METHOD PRIVATE CheckCanHomeTransferArm
VAR_IN_OUT
    stSDS : ST_SDS;
    stSDSP : ST_SDSPersistent;
END_VAR

stSDS.bSuccess := FALSE;

stSDS.sStatusMsg := 'Checking if transfer arm can be homed.';

InitHomeTransferArm(
    stSDS := stSDS
);

stSDS.bSuccess := TRUE;
END_METHOD


METHOD PRIVATE CheckCanLoadArmFromGarage
VAR_IN_OUT
    stSDS : ST_SDS;
    stSDSP : ST_SDSPersistent;
END_VAR

stSDS.bSuccess := FALSE;

stSDS.sStatusMsg := 'Checking if there is an open slot in the transfer arm and at least one full slot in the garage.';

CheckCanDo2Criteria(
    bCanDo := stSDS.bSuccess,
    bCantDo := stSDS.bError,
    sErrorMsg := stSDS.sErrorMsg,
    b1 := stSDS.bGarageUnloadable,
    b2 := stSDS.bTransferArmLoadable,
    sErrorMsgTF := 'The transfer arm is currently full and cannot be used to remove a sample from the garage.',
    sErrorMsgFT := 'The garage is currently empty and therefore no samples can be removed.',
    sErrorMsgFF := 'The garage is currently empty and the transfer arm is full. Therefore, no samples can be removed.'
);
END_METHOD


METHOD PRIVATE CheckCanLoadDiffractometerFromArm
VAR_IN_OUT
    stSDS : ST_SDS;
    stSDSP : ST_SDSPersistent;
END_VAR

stSDS.bSuccess := FALSE;

stSDS.sStatusMsg := 'Checking if the diffractometer slot is open and if the transfer arm is carrying a sample.';

CheckCanDo2Criteria(
    bCanDo := stSDS.bSuccess,
    bCantDo := stSDS.bError,
    sErrorMsg := stSDS.sErrorMsg,
    b1 := stSDS.bDiffractometerLoadable,
    b2 := stSDS.bTransferArmUnloadable,
    sErrorMsgTF := 'The transfer arm is currently empty and cannot be used to place a sample in the diffractometer.',
    sErrorMsgFT := 'The diffractometer already has a sample in it.',
    sErrorMsgFF := 'The diffractoemter already has a sample and the transfer arm is empty.'
);
END_METHOD


METHOD PRIVATE CheckCanLoadUnloadGarageFromPort
VAR_IN_OUT
    stSDS : ST_SDS;
    stSDSP : ST_SDSPersistent;
END_VAR

stSDS.bSuccess := FALSE;

stSDS.sStatusMsg := 'Checking if the garage can be loaded or unloaded from the port.';

stSDS.bSuccess := TRUE;
END_METHOD


METHOD PRIVATE CheckCanManualControl
VAR_IN_OUT
    stSDS : ST_SDS;
    stSDSP : ST_SDSPersistent;
END_VAR

stSDS.bSuccess := FALSE;

stSDS.sStatusMsg := 'Checking if we can switch to manual control.';

stSDS.bSuccess := TRUE;
END_METHOD


METHOD PRIVATE CheckCanUnloadArmToGarage
VAR_IN_OUT
    stSDS : ST_SDS;
    stSDSP : ST_SDSPersistent;
END_VAR

stSDS.bSuccess := FALSE;

stSDS.sStatusMsg := 'Checking if there is an open slot in the garage and if the transfer arm is carrying a sample.';

CheckCanDo2Criteria(
    bCanDo := stSDS.bSuccess,
    bCantDo := stSDS.bError,
    sErrorMsg := stSDS.sErrorMsg,
    b1 := stSDS.bGarageLoadable,
    b2 := stSDS.bTransferArmUnloadable,
    sErrorMsgTF := 'The transfer arm is currently empty and cannot be used to load sample into the garage.',
    sErrorMsgFT := 'The garage is currently full and therefore no samples can be loaded into it.',
    sErrorMsgFF := 'The garage is currently full and the transfer arm is empty.'
);
END_METHOD


METHOD PRIVATE CheckCanUnloadDiffractometerToArm
VAR_IN_OUT
    stSDS : ST_SDS;
    stSDSP : ST_SDSPersistent;
END_VAR

stSDS.bSuccess := FALSE;

stSDS.sStatusMsg := 'Checking if the diffractometer slot is full and if the transfer arm is empty.';

CheckCanDo2Criteria(
    bCanDo := stSDS.bSuccess,
    bCantDo := stSDS.bError,
    sErrorMsg := stSDS.sErrorMsg,
    b1 := stSDS.bDiffractometerUnloadable,
    b2 := stSDS.bTransferArmLoadable,
    sErrorMsgTF := 'The transfer arm is currently full and cannot be used to unload a sample from the diffractometer.',
    sErrorMsgFT := 'The diffractometer does not have a sample in it.',
    sErrorMsgFF := 'The diffractometeris empty and the transfer arm is full.'
);
END_METHOD


METHOD PRIVATE ConfirmDiffractometerExtraction
VAR_IN_OUT
    stSDS : ST_SDS;
END_VAR

stSDS.bSuccess := FALSE;

stSDS.sStatusMsg := 'Moving transfer arm back a few mm. Please confirm the sample is held by the diffractometer and then click "proceed". If the sample is still in the transfer arm, click "retry" to go back to fine adjustment.';

SetPositionStateWaitForArrivalQuitIfError(
    eStateGet := stSDS.eTransferArmHStateGet,
    stMotionStage := stSDS.stTransferArmHStage,
    eStateSet := stSDS.eTransferArmHStateSet,
    eEnumSet := E_SDSTransferArmHStates.CONFIRM_DIFF_EXTRACTION,
    bError := stSDS.bError,
    sErrorMsg := stSDS.sErrorMsg,
    bArrived => stSDS.bSuccess
);
END_METHOD


METHOD PRIVATE ConfirmDiffractometerInsertion
VAR_IN_OUT
    stSDS : ST_SDS;
END_VAR

stSDS.bSuccess := FALSE;

stSDS.sStatusMsg := 'Moving transfer arm back a few mm. Please confirm the sample is held by the diffractometer and then click "proceed". If the sample is still in the transfer arm, click "retry" to go back to fine adjustment.';

SetPositionStateWaitForArrivalQuitIfError(
    eStateGet := stSDS.eTransferArmHStateGet,
    stMotionStage := stSDS.stTransferArmHStage,
    eStateSet := stSDS.eTransferArmHStateSet,
    eEnumSet := E_SDSTransferArmHStates.CONFIRM_DIFF_INSERTION,
    bError := stSDS.bError,
    sErrorMsg := stSDS.sErrorMsg,
    bArrived => stSDS.bSuccess
);
END_METHOD


METHOD PRIVATE ConfirmExtraction
VAR_IN_OUT
    stSDS : ST_SDS;
END_VAR

stSDS.bSuccess := FALSE;

stSDS.sStatusMsg := 'Moving transfer arm back a few mm. Please confirm the sample is held by the arm and then click "proceed". If the sample is still in the holder, click "retry" to go back to fine adjustment.';

SetPositionStateWaitForArrivalQuitIfError(
    eStateGet := stSDS.eTransferArmHStateGet,
    stMotionStage := stSDS.stTransferArmHStage,
    eStateSet := stSDS.eTransferArmHStateSet,
    eEnumSet := E_SDSTransferArmHStates.CONFIRM_GARAGE_EXTRACTION,
    bError := stSDS.bError,
    sErrorMsg := stSDS.sErrorMsg,
    bArrived => stSDS.bSuccess
);
END_METHOD


METHOD PRIVATE ConfirmGarageFreeToRotate
VAR_IN_OUT
    stSDS : ST_SDS;
    stSDSP : ST_SDSPersistent;
END_VAR
VAR_INST
    tonHoldDelay : TON;
END_VAR

// Missing handling for erroring encoder.

tonHoldDelay(
    IN := stSDS.stGarageYStage.Axis.NcToPlc.ActPos >= stSDSP.fGarageHeightSafeFromCollision,
    PT := T#1s
);

stSDS.bGarageAboveCollisionHeight := tonHoldDelay.Q;
END_METHOD


METHOD PRIVATE ConfirmInsertion
VAR_IN_OUT
    stSDS : ST_SDS;
END_VAR

stSDS.bSuccess := FALSE;

stSDS.sStatusMsg := 'Moving transfer arm back a few mm. Please confirm the sample is held by the garage and then click "proceed". If the sample is still in the transfer arm, click "retry" to go back to fine adjustment.';

SetPositionStateWaitForArrivalQuitIfError(
    eStateGet := stSDS.eTransferArmHStateGet,
    stMotionStage := stSDS.stTransferArmHStage,
    eStateSet := stSDS.eTransferArmHStateSet,
    eEnumSet := E_SDSTransferArmHStates.CONFIRM_GARAGE_INSERTION,
    bError := stSDS.bError,
    sErrorMsg := stSDS.sErrorMsg,
    bArrived => stSDS.bSuccess
);
END_METHOD


METHOD PRIVATE ConfirmVacuumValveOpen
VAR_IN_OUT
    stSDS : ST_SDS;
END_VAR

stSDS.sStatusMsg := 'Verifying that the vacuum valve between SDS and Diff is open.';

stSDS.bSuccess := GVL_Interface.QRIX_VAC_VGC_03_OPEN_LIMIT_SWITCH AND
    NOT GVL_Interface.QRIX_VAC_VGC_03_CLOSED_LIMIT_SWITCH;
END_METHOD


METHOD PRIVATE ExtendPrerotateTransferArmForLoading
VAR_IN_OUT
    stSDS : ST_SDS;
END_VAR
VAR
    bHArrived : BOOL;
    bRArrived : BOOL;
END_VAR

stSDS.bSuccess := FALSE;

stSDS.sStatusMsg := 'Moving transfer arm to nominal sample loading position and pre-rotating to allow full rotation for screwing in sample.';

SetPositionStateWaitForArrivalQuitIfError(
    eStateGet := stSDS.eTransferArmHStateGet,
    stMotionStage := stSDS.stTransferArmHStage,
    eStateSet := stSDS.eTransferArmHStateSet,
    eEnumSet := E_SDSTransferArmHStates.GARAGE_SAMPLE_INSERTION,
    bError := stSDS.bError,
    sErrorMsg := stSDS.sErrorMsg,
    bArrived => bHArrived
);

SetPositionStateWaitForArrivalQuitIfError(
    eStateGet := stSDS.eTransferArmRStateGet,
    stMotionStage := stSDS.stTransferArmRStage,
    eStateSet := stSDS.eTransferArmRStateSet,
    eEnumSet := E_SDSTransferArmRStates.PREROTATE_SAMPLE_INSERTION,
    bError := stSDS.bError,
    sErrorMsg := stSDS.sErrorMsg,
    bArrived => bRArrived
);

IF bHArrived AND bRArrived THEN
    stSDS.bSuccess := TRUE;
END_IF
END_METHOD


METHOD PRIVATE ExtendTransferArmForDiffractometerExtraction
VAR_IN_OUT
    stSDS : ST_SDS;
END_VAR

stSDS.bSuccess := FALSE;

stSDS.sStatusMsg := 'Moving transfer arm to nominal sample unloading position for diffractometer.';

SetPositionStateWaitForArrivalQuitIfError(
    eStateGet := stSDS.eTransferArmHStateGet,
    stMotionStage := stSDS.stTransferArmHStage,
    eStateSet := stSDS.eTransferArmHStateSet,
    eEnumSet := E_SDSTransferArmHStates.DIFF_SAMPLE_EXTRACTION,
    bError := stSDS.bError,
    sErrorMsg := stSDS.sErrorMsg,
    bArrived => stSDS.bSuccess
);
END_METHOD


METHOD PRIVATE ExtendTransferArmForDiffractometerInsertion
VAR_IN_OUT
    stSDS : ST_SDS;
END_VAR

stSDS.bSuccess := FALSE;

stSDS.sStatusMsg := 'Moving transfer arm to nominal sample loading position for diffractometer.';

SetPositionStateWaitForArrivalQuitIfError(
    eStateGet := stSDS.eTransferArmHStateGet,
    stMotionStage := stSDS.stTransferArmHStage,
    eStateSet := stSDS.eTransferArmHStateSet,
    eEnumSet := E_SDSTransferArmHStates.DIFF_SAMPLE_INSERTION,
    bError := stSDS.bError,
    sErrorMsg := stSDS.sErrorMsg,
    bArrived => stSDS.bSuccess
);
END_METHOD


METHOD PRIVATE ExtendTransferArmForExtraction
VAR_IN_OUT
    stSDS : ST_SDS;
END_VAR

stSDS.bSuccess := FALSE;

stSDS.sStatusMsg := 'Moving transfer arm to nominal sample extraction position for garage.';

SetPositionStateWaitForArrivalQuitIfError(
    eStateGet := stSDS.eTransferArmHStateGet,
    stMotionStage := stSDS.stTransferArmHStage,
    eStateSet := stSDS.eTransferArmHStateSet,
    eEnumSet := E_SDSTransferArmHStates.GARAGE_SAMPLE_REMOVAL,
    bError := stSDS.bError,
    sErrorMsg := stSDS.sErrorMsg,
    bArrived => stSDS.bSuccess
);
END_METHOD


METHOD PRIVATE ExtendTransferArmForInsertion
VAR_IN_OUT
    stSDS : ST_SDS;
END_VAR
VAR
    bHArrived : BOOL;
    bRArrived : BOOL;
END_VAR

stSDS.bSuccess := FALSE;

stSDS.sStatusMsg := 'Moving transfer arm to nominal sample loading position for garage.';

SetPositionStateWaitForArrivalQuitIfError(
    eStateGet := stSDS.eTransferArmHStateGet,
    stMotionStage := stSDS.stTransferArmHStage,
    eStateSet := stSDS.eTransferArmHStateSet,
    eEnumSet := E_SDSTransferArmHStates.GARAGE_SAMPLE_INSERTION,
    bError := stSDS.bError,
    sErrorMsg := stSDS.sErrorMsg,
    bArrived => stSDS.bSuccess
);
END_METHOD


METHOD PRIVATE FineAdjustment
VAR_IN_OUT
    stSDS : ST_SDS;
END_VAR

stSDS.sStatusMsg := 'Use the individual motor control to do fine adjustment. Click "proceed" to move to the next step.';
END_METHOD


METHOD PRIVATE GarageFaceTransferArm
VAR_IN_OUT
    stSDS : ST_SDS;
END_VAR
VAR
    bYArrived : BOOL;
    bRArrived : BOOL;
END_VAR

stSDS.bSuccess := FALSE;

stSDS.sStatusMsg := 'Facing garage towards the transfer arm.';

stSDS.eFaceState := E_SDSFaceState.FACE_TRANSFER_ARM;

SetPositionStateWaitForArrivalQuitIfError(
    eStateGet := stSDS.eGarageRStateGet,
    stMotionStage := stSDS.stGarageRStage,
    eStateSet := stSDS.eGarageRStateSet,
    eEnumSet := stSDS.eSelectedGarageSlot,
    bError := stSDS.bError,
    sErrorMsg := stSDS.sErrorMsg,
    bArrived => stSDS.bSuccess
);
END_METHOD


METHOD PRIVATE HoldThenClear
VAR_IN_OUT
    b1 : BOOL;
END_VAR
VAR_INPUT
    tHoldDuration : TIME := T#1s;
END_VAR
VAR_INST
    tonHoldTimer : TON;
END_VAR

tonHoldTimer(IN := b1, PT := tHoldDuration);

IF tonHoldTimer.Q THEN
    b1 := FALSE;
END_IF
END_METHOD


METHOD PRIVATE HomeGarage
VAR_IN_OUT
    stSDS : ST_SDS;
END_VAR

stSDS.bSuccess := FALSE;

stSDS.sStatusMsg := 'Homing the garage.';

IF stSDS.stGarageRStage.bError THEN
    stSDS.bError := TRUE;
    stSDS.sErrorMsg := 'Garage rotational stage has an active error. Aborting sequence.';
END_IF

HomeStateMachine(
    eHomingState := stSDS.eGarageRHomingState,
    stMotionStage := stSDS.stGarageRStage,
    bError => stSDS.bError,
    sErrorMsg => stSDS.sErrorMsg
);

IF stSDS.eGarageRHomingState = E_SDSHomingState.HOMED THEN
    stSDS.bSuccess := TRUE;
END_IF
END_METHOD


METHOD PRIVATE HomeStateMachine
VAR_IN_OUT
    eHomingState : E_SDSHomingState;
    stMotionStage : ST_MotionStage;
END_VAR
VAR_OUTPUT
    bError : BOOL;
    sErrorMsg : T_MaxString;
END_VAR

IF stMotionStage.bHome AND F_Limit(
    fVal := stMotionStage.Axis.NcToPlc.ActPos,
    fLLim := -0.01,
    fHLim := 0.01,
    bInclusive := TRUE) THEN
    eHomingState := E_SDSHomingState.HOMED;
END_IF

CASE eHomingState OF
    E_SDSHomingState.INIT:
        eHomingState := E_SDSHomingState.WAIT_NOT_BUSY;
    E_SDSHomingState.WAIT_NOT_BUSY:
        IF NOT stMotionStage.bBusy THEN
            eHomingState := E_SDSHomingState.TRIGGER_HOMING;
        END_IF
    E_SDSHomingState.TRIGGER_HOMING:
        stMotionStage.bHomeCmd := TRUE;
        IF stMotionStage.nCommand = E_EpicsMotorCmd.HOME AND stMotionStage.bBusy THEN
            eHomingState := E_SDSHomingState.WAIT_FOR_HOMED;
        END_IF
    E_SDSHomingState.WAIT_FOR_HOMED:
        IF stMotionStage.bDone THEN
            eHomingState := E_SDSHomingState.HOMED;
        END_IF
ELSE
    bError := TRUE;
    sErrorMsg := 'Homing sequence triggered an unknown state. Aborting sequence.';
END_CASE
END_METHOD


METHOD PRIVATE HomeTransferArm
VAR_IN_OUT
    stSDS : ST_SDS;
END_VAR

stSDS.bSuccess := FALSE;

stSDS.sStatusMsg := 'Homing the transfer arm.';

IF stSDS.stTransferArmHStage.bError THEN
    stSDS.bError := TRUE;
    stSDS.sErrorMsg := 'Transfer arm horizontal stage has an active error. Aborting sequence.';
END_IF

IF stSDS.stTransferArmRStage.bError THEN
    stSDS.bError := TRUE;
    stSDS.sErrorMsg := 'Transfer arm rotational stage has an active error. Aborting sequence.';
END_IF

HomeStateMachine(
    eHomingState := stSDS.eTransferArmHHomingState,
    stMotionStage := stSDS.stTransferArmHStage,
    bError => stSDS.bError,
    sErrorMsg => stSDS.sErrorMsg
);

HomeStateMachine(
    eHomingState := stSDS.eTransferArmRHomingState,
    stMotionStage := stSDS.stTransferArmRStage,
    bError => stSDS.bError,
    sErrorMsg => stSDS.sErrorMsg
);

IF stSDS.eTransferArmHHomingState = E_SDSHomingState.HOMED AND
   stSDS.eTransferArmRHomingState = E_SDSHomingState.HOMED THEN
    stSDS.bSuccess := TRUE;
END_IF
END_METHOD


METHOD PRIVATE InitHomeGarage
VAR_IN_OUT
    stSDS : ST_SDS;
END_VAR

stSDS.eGarageRHomingState := E_SDSHomingState.INIT;
END_METHOD


METHOD PRIVATE InitHomeTransferArm
VAR_IN_OUT
    stSDS : ST_SDS;
END_VAR

stSDS.eTransferArmHHomingState := E_SDSHomingState.INIT;
stSDS.eTransferArmRHomingState := E_SDSHomingState.INIT;
END_METHOD


METHOD PRIVATE InitRotateGarageForClearance
VAR_IN_OUT
    stSDS : ST_SDS;
    stSDSP : ST_SDSPersistent;
END_VAR

stSDS.fGarageRotationClearancePos := stSDS.stGarageRStage.Axis.NcToPlc.ActPos + stSDSP.fGarageRotationClearanceOffset;
END_METHOD


METHOD PRIVATE InitSelectGarageSlotForLoading
VAR_IN_OUT
    stSDS : ST_SDS;
    stSDSP : ST_SDSPersistent;
END_VAR

FOR nIndex := E_SDSGarageYStates.T1 TO E_SDSGarageYStates.B4 BY 1 DO
    CASE stSDSP.astGarageSlot[nIndex].eState OF
        E_SampleSlotStates.EMPTY:
            stSDS.eSelectedGarageSlot := nIndex;
    END_CASE
END_FOR

IF nIndex > E_SDSGarageYStates.B4 THEN
    stSDS.bError := TRUE;
    stSDS.sErrorMsg := 'There are no empty slots in the garage to load a sample to.';
END_IF
END_METHOD


METHOD PRIVATE InitSelectGarageSlotForRemoval
VAR_IN_OUT
    stSDS : ST_SDS;
    stSDSP : ST_SDSPersistent;
END_VAR

FOR nIndex := E_SDSGarageYStates.T1 TO E_SDSGarageYStates.B4 BY 1 DO
    CASE stSDSP.astGarageSlot[nIndex].eState OF
        E_SampleSlotStates.FULL:
            stSDS.eSelectedGarageSlot := nIndex;
    END_CASE
END_FOR

IF nIndex > E_SDSGarageYStates.B4 THEN
    stSDS.bError := TRUE;
    stSDS.sErrorMsg := 'There are no full slots in the garage to extract a sample from.';
END_IF
END_METHOD


METHOD PRIVATE LoadArmFromGarage
VAR_IN_OUT
    stSDS : ST_SDS;
    stSDSP : ST_SDSPersistent;
END_VAR

CASE stSDS.eSeqState OF
    E_SDSSeqState.Inactive:
        stSDS.eSeqState := E_SDSSeqState.Home_Transfer_Arm;
    E_SDSSeqState.Home_Transfer_Arm:
        HomeTransferArm(
            stSDS := stSDS
        );
        IF stSDS.bSuccess THEN
            stSDS.eSeqState := E_SDSSeqState.Check_Garage_Height;
        END_IF
    E_SDSSeqState.Check_Garage_Height:
        IF stSDS.bGarageAboveCollisionHeight THEN
            stSDS.eSeqState := E_SDSSeqState.Home_Garage;
        ELSE
            stSDS.eSeqState := E_SDSSeqState.Manually_Rotate_Garage_for_Clearance_to_Raise;
        END_IF
    E_SDSSeqState.Manually_Rotate_Garage_for_Clearance_to_Raise:
        RotateGarageForClearanceManual(
            stSDS := stSDS
        );
        IF stSDS.stUISelect.bProceed THEN
            stSDS.eSeqState := E_SDSSeqState.Retract_Garage_1;
        END_IF
    E_SDSSeqState.Retract_Garage_1:
        RetractGarage(
            stSDS := stSDS
        );
        IF stSDS.bSuccess THEN
            stSDS.eSeqState := E_SDSSeqState.Home_Garage;
        END_IF
    E_SDSSeqState.Home_Garage:
        HomeGarage(
            stSDS := stSDS
        );
        IF stSDS.bSuccess THEN
            stSDS.eSeqState := E_SDSSeqState.Select_Garage_Slot_for_Removal;
        END_IF
    E_SDSSeqState.Select_Garage_Slot_for_Removal:
        SelectGarageSlotForRemoval(
            stSDS := stSDS,
            stSDSP := stSDSP
        );
        IF stSDS.bSuccess THEN
            stSDS.eSeqState := E_SDSSeqState.Garage_Face_Transfer_Arm;
        END_IF
    E_SDSSeqState.Garage_Face_Transfer_Arm:
        GarageFaceTransferArm(
            stSDS := stSDS
        );
        IF stSDS.bSuccess THEN
            stSDS.eSeqState := E_SDSSeqState.Rotate_Garage_for_Clearance_to_Lower;
        END_IF
    E_SDSSeqState.Rotate_Garage_for_Clearance_to_Lower:
        RotateGarageForClearance(
            stSDS := stSDS
        );
        IF stSDS.bSuccess THEN
            stSDS.eSeqState := E_SDSSeqState.Move_Garage_to_Slot_Height;
        END_IF
    E_SDSSeqState.Move_Garage_to_Slot_Height:
        MoveGarageToSlotHeight(
            stSDS := stSDS
        );
        IF stSDS.bSuccess THEN
            stSDS.eSeqState := E_SDSSeqState.Prerotate_Transfer_Arm_for_Extraction;
        END_IF
    E_SDSSeqState.Prerotate_Transfer_Arm_for_Extraction:
        PrerotateTransferArmForExtraction(
            stSDS := stSDS
        );
        IF stSDS.bSuccess THEN
            stSDS.eSeqState := E_SDSSeqState.Extend_Transfer_Arm_for_Extraction;
        END_IF
    E_SDSSeqState.Extend_Transfer_Arm_for_Extraction:
        ExtendTransferArmForExtraction(
            stSDS := stSDS
        );
        IF stSDS.bSuccess THEN
            stSDS.eSeqState := E_SDSSeqState.Screw_in_Half_Turn;
        END_IF
    E_SDSSeqState.Screw_in_Half_Turn:
        ScrewInHalfTurn(
            stSDS := stSDS
        );
        IF stSDS.bSuccess THEN
            stSDS.eSeqState := E_SDSSeqState.Fine_Adjustment;
        END_IF
    E_SDSSeqState.Fine_Adjustment:
        FineAdjustment(
            stSDS := stSDS
        );
        IF stSDS.stUISelect.bProceed THEN
            stSDS.eSeqState := E_SDSSeqState.Unscrew_Sample_from_Garage;
        END_IF
    E_SDSSeqState.Unscrew_Sample_from_Garage:
        UnscrewSampleFromGarage(
            stSDS := stSDS
        );
        IF stSDS.bSuccess THEN
            stSDS.eSeqState := E_SDSSeqState.Confirm_Extraction;
        END_IF
    E_SDSSeqState.Confirm_Extraction:
        ConfirmExtraction(
            stSDS := stSDS
        );
        IF stSDS.bSuccess AND stSDS.stUISelect.bProceed THEN
            stSDS.eSeqState := E_SDSSeqState.Update_Sample_Database;
        ELSIF stSDS.stUISelect.bRetry THEN
            stSDS.eSeqState := E_SDSSeqState.Fine_Adjustment;
        END_IF
    E_SDSSeqState.Update_Sample_Database:
        UpdateSampleLocationDatabaseGarageToArm(
            stSDS := stSDS,
            stSDSP := stSDSP
        );
        IF stSDS.bSuccess OR stSDS.stUISelect.bProceed THEN
            stSDS.eSeqState := E_SDSSeqState.Retract_Transfer_Arm;
        END_IF
    E_SDSSeqState.Retract_Transfer_Arm:
        HomeTransferArm(
            stSDS := stSDS
        );
        IF stSDS.bSuccess THEN
            stSDS.eSeqState := E_SDSSeqState.Rotate_Garage_for_Clearance_to_Raise;
        END_IF
    E_SDSSeqState.Rotate_Garage_for_Clearance_to_Raise:
        RotateGarageForClearance(
            stSDS := stSDS
        );
        IF stSDS.bSuccess THEN
            stSDS.eSeqState := E_SDSSeqState.Retract_Garage_2;
        END_IF
    E_SDSSeqState.Retract_Garage_2:
        RetractGarage(
            stSDS := stSDS
        );
        IF stSDS.bSuccess THEN
            stSDS.eSeqState := E_SDSSeqState.Return_Garage_to_Home;
        END_IF
    E_SDSSeqState.Return_Garage_to_Home:
        HomeGarage(
            stSDS := stSDS
        );
        IF stSDS.bSuccess THEN
            stSDS.eState := E_SDSState.Standby;
        END_IF
END_CASE
END_METHOD


METHOD PRIVATE LoadDiffractometerFromArm
VAR_IN_OUT
    stSDS : ST_SDS;
    stSDSP : ST_SDSPersistent;
END_VAR

CASE stSDS.eSeqState OF
    E_SDSSeqState.Inactive:
        stSDS.eSeqState := E_SDSSeqState.Home_Transfer_Arm;
    E_SDSSeqState.Home_Transfer_Arm:
        HomeTransferArm(
            stSDS := stSDS
        );
        IF stSDS.bSuccess THEN
            stSDS.eSeqState := E_SDSSeqState.Check_Garage_Height;
        END_IF
    E_SDSSeqState.Check_Garage_Height:
        IF stSDS.bGarageAboveCollisionHeight THEN
            stSDS.eSeqState := E_SDSSeqState.Home_Garage;
        ELSE
            stSDS.eSeqState := E_SDSSeqState.Manually_Rotate_Garage_for_Clearance_to_Raise;
        END_IF
    E_SDSSeqState.Manually_Rotate_Garage_for_Clearance_to_Raise:
        RotateGarageForClearanceManual(
            stSDS := stSDS
        );
        IF stSDS.stUISelect.bProceed THEN
            stSDS.eSeqState := E_SDSSeqState.Retract_Garage_1;
        END_IF
    E_SDSSeqState.Retract_Garage_1:
        RetractGarage(
            stSDS := stSDS
        );
        IF stSDS.bSuccess THEN
            stSDS.eSeqState := E_SDSSeqState.Home_Garage;
        END_IF
    E_SDSSeqState.Home_Garage:
        HomeGarage(
            stSDS := stSDS
        );
        IF stSDS.bSuccess THEN
            stSDS.eSeqState := E_SDSSeqState.Move_Diffractometer_to_Load_Unload_Position;
        END_IF
    E_SDSSeqState.Move_Diffractometer_to_Load_Unload_Position:
        MoveDiffractometerToLoadUnloadPosition(
            stSDS := stSDS
        );
        IF stSDS.bSuccess THEN
            stSDS.eSeqState := E_SDSSeqState.Confirm_Vacuum_Valve_Open;
        END_IF
    E_SDSSeqState.Confirm_Vacuum_Valve_Open:
        ConfirmVacuumValveOpen(
            stSDS := stSDS
        );
        IF stSDS.bSuccess THEN
            stSDS.eSeqState := E_SDSSeqState.Prerotate_Transfer_Arm_for_Insertion;
        END_IF
    E_SDSSeqState.Prerotate_Transfer_Arm_for_Insertion:
        PrerotateTransferArmForInsertion(
            stSDS := stSDS
        );
        IF stSDS.bSuccess THEN
            stSDS.eSeqState := E_SDSSeqState.Extend_Transfer_Arm_for_Diffractometer_Insertion;
        END_IF
    E_SDSSeqState.Extend_Transfer_Arm_for_Diffractometer_Insertion:
        ExtendTransferArmForDiffractometerInsertion(
            stSDS := stSDS
        );
        IF stSDS.bSuccess THEN
            stSDS.eSeqState := E_SDSSeqState.Fine_Adjustment;
        END_IF
    E_SDSSeqState.Fine_Adjustment:
        FineAdjustment(
            stSDS := stSDS
        );
        IF stSDS.stUISelect.bProceed THEN
            stSDS.eSeqState := E_SDSSeqState.Screw_Sample_into_Diffractometer;
        END_IF
    E_SDSSeqState.Screw_Sample_into_Diffractometer:
        ScrewSampleIntoDiffractometer(
            stSDS := stSDS
        );
        IF stSDS.bSuccess THEN
            stSDS.eSeqState := E_SDSSeqState.Confirm_Diffractometer_Insertion;
        END_IF
    E_SDSSeqState.Confirm_Diffractometer_Insertion:
        ConfirmDiffractometerInsertion(
            stSDS := stSDS
        );
        IF stSDS.bSuccess AND stSDS.stUISelect.bProceed THEN
            stSDS.eSeqState := E_SDSSeqState.Update_Sample_Database;
        ELSIF stSDS.stUISelect.bRetry THEN
            stSDS.eSeqState := E_SDSSeqState.Fine_Adjustment;
        END_IF
    E_SDSSeqState.Update_Sample_Database:
        UpdateSampleLocationDatabaseDiffToArm(
            stSDS := stSDS,
            stSDSP := stSDSP
        );
        IF stSDS.bSuccess OR stSDS.stUISelect.bProceed THEN
            stSDS.eSeqState := E_SDSSeqState.Retract_Transfer_Arm;
        END_IF
    E_SDSSeqState.Retract_Transfer_Arm:
        HomeTransferArm(
            stSDS := stSDS
        );
        IF stSDS.bSuccess THEN
            stSDS.eSeqState := E_SDSSeqState.Rotate_Garage_for_Clearance_to_Raise;
        END_IF
END_CASE
END_METHOD


METHOD PRIVATE LoadUnloadGarageFromPort
VAR_IN_OUT
    stSDS : ST_SDS;
    stSDSP : ST_SDSPersistent;
END_VAR
END_METHOD


METHOD PRIVATE ManualControl
VAR_IN_OUT
    stSDS : ST_SDS;
    stSDSP : ST_SDSPersistent;
END_VAR
END_METHOD


METHOD PRIVATE MoveDiffractometerToLoadUnloadPosition
VAR_IN_OUT
    stSDS : ST_SDS;
END_VAR
VAR
    bXArrived : BOOL;
    bYArrived : BOOL;
    bZArrived : BOOL;
    b2ThetaYArrived : BOOL;
    bPhiArrived : BOOL;
    bChiArrived : BOOL;
    b2ThetaArrived : BOOL;
    bThetaArrived : BOOL;
END_VAR

stSDS.bSuccess := FALSE;

stSDS.sStatusMsg := 'Moving the diffractometer to load/unload position.';

SetPositionStateWaitForArrivalQuitIfError(
    eStateGet := stSDS.eDiffXStateGet,
    stMotionStage := stSDS.stDiffXStage,
    eStateSet := stSDS.eDiffXStateSet,
    eEnumSet := E_DiffState.TRANSFER_ARM_INTERFACE,
    bError := stSDS.bError,
    sErrorMsg := stSDS.sErrorMsg,
    bArrived => bXArrived
);

SetPositionStateWaitForArrivalQuitIfError(
    eStateGet := stSDS.eDiffYStateGet,
    stMotionStage := stSDS.stDiffYStage,
    eStateSet := stSDS.eDiffYStateSet,
    eEnumSet := E_DiffState.TRANSFER_ARM_INTERFACE,
    bError := stSDS.bError,
    sErrorMsg := stSDS.sErrorMsg,
    bArrived => bYArrived
);

SetPositionStateWaitForArrivalQuitIfError(
    eStateGet := stSDS.eDiffZStateGet,
    stMotionStage := stSDS.stDiffZStage,
    eStateSet := stSDS.eDiffZStateSet,
    eEnumSet := E_DiffState.TRANSFER_ARM_INTERFACE,
    bError := stSDS.bError,
    sErrorMsg := stSDS.sErrorMsg,
    bArrived => bZArrived
);

SetPositionStateWaitForArrivalQuitIfError(
    eStateGet := stSDS.eDiff2ThetaYStateGet,
    stMotionStage := stSDS.stDiff2ThetaYStage,
    eStateSet := stSDS.eDiff2ThetaYStateSet,
    eEnumSet := E_DiffState.TRANSFER_ARM_INTERFACE,
    bError := stSDS.bError,
    sErrorMsg := stSDS.sErrorMsg,
    bArrived => b2ThetaYArrived
);

SetPositionStateWaitForArrivalQuitIfError(
    eStateGet := stSDS.eDiffPhiStateGet,
    stMotionStage := stSDS.stDiffPhiStage,
    eStateSet := stSDS.eDiffPhiStateSet,
    eEnumSet := E_DiffState.TRANSFER_ARM_INTERFACE,
    bError := stSDS.bError,
    sErrorMsg := stSDS.sErrorMsg,
    bArrived => bPhiArrived
);

SetPositionStateWaitForArrivalQuitIfError(
    eStateGet := stSDS.eDiffChiStateGet,
    stMotionStage := stSDS.stDiffChiStage,
    eStateSet := stSDS.eDiffChiStateSet,
    eEnumSet := E_DiffState.TRANSFER_ARM_INTERFACE,
    bError := stSDS.bError,
    sErrorMsg := stSDS.sErrorMsg,
    bArrived => bChiArrived
);

SetPositionStateWaitForArrivalQuitIfError(
    eStateGet := stSDS.eDiff2ThetaStateGet,
    stMotionStage := stSDS.stDiff2ThetaStage,
    eStateSet := stSDS.eDiff2ThetaStateSet,
    eEnumSet := E_DiffState.TRANSFER_ARM_INTERFACE,
    bError := stSDS.bError,
    sErrorMsg := stSDS.sErrorMsg,
    bArrived => b2ThetaArrived
);

SetPositionStateWaitForArrivalQuitIfError(
    eStateGet := stSDS.eDiffThetaStateGet,
    stMotionStage := stSDS.stDiffThetaStage,
    eStateSet := stSDS.eDiffThetaStateSet,
    eEnumSet := E_DiffState.TRANSFER_ARM_INTERFACE,
    bError := stSDS.bError,
    sErrorMsg := stSDS.sErrorMsg,
    bArrived => bThetaArrived
);

IF bXArrived AND
   bYArrived AND
   bZArrived AND
   b2ThetaYArrived AND
   bPhiArrived AND
   bChiArrived AND
   b2ThetaArrived AND
   bThetaArrived THEN
    stSDS.bSuccess := TRUE;
END_IF
END_METHOD


METHOD PRIVATE MoveGarageToSlotHeight
VAR_IN_OUT
    stSDS : ST_SDS;
END_VAR

stSDS.bSuccess := FALSE;

stSDS.sStatusMsg := 'Moving garage to selected slot height.';

SetPositionStateWaitForArrivalQuitIfError(
    eStateGet := stSDS.eGarageYStateGet,
    stMotionStage := stSDS.stGarageYStage,
    eStateSet := stSDS.eGarageYStateSet,
    eEnumSet := stSDS.eSelectedGarageSlot,
    bError := stSDS.bError,
    sErrorMsg := stSDS.sErrorMsg,
    bArrived => stSDS.bSuccess
);
END_METHOD


METHOD PRIVATE MoveToGarageSlotFaceTransferArm
VAR_IN_OUT
    stSDS : ST_SDS;
END_VAR
VAR
    bYArrived : BOOL;
    bRArrived : BOOL;
END_VAR

stSDS.bSuccess := FALSE;

stSDS.sStatusMsg := 'Moving garage to selected slot and facing it towards transfer arm.';

stSDS.eFaceState := E_SDSFaceState.FACE_TRANSFER_ARM;

SetPositionStateWaitForArrivalQuitIfError(
    eStateGet := stSDS.eGarageYStateGet,
    stMotionStage := stSDS.stGarageYStage,
    eStateSet := stSDS.eGarageYStateSet,
    eEnumSet := stSDS.eSelectedGarageSlot,
    bError := stSDS.bError,
    sErrorMsg := stSDS.sErrorMsg,
    bArrived => bYArrived
);

SetPositionStateWaitForArrivalQuitIfError(
    eStateGet := stSDS.eGarageRStateGet,
    stMotionStage := stSDS.stGarageRStage,
    eStateSet := stSDS.eGarageRStateSet,
    eEnumSet := stSDS.eSelectedGarageSlot,
    bError := stSDS.bError,
    sErrorMsg := stSDS.sErrorMsg,
    bArrived => bRArrived
);

IF bYArrived AND bRArrived THEN
    stSDS.bSuccess := TRUE;
END_IF
END_METHOD


METHOD PRIVATE PrerotateTransferArmForExtraction
VAR_IN_OUT
    stSDS : ST_SDS;
END_VAR

stSDS.bSuccess := FALSE;

stSDS.sStatusMsg := 'Pre-rotating transfer arm to allow full rotation for unscrewing the sample.';

SetPositionStateWaitForArrivalQuitIfError(
    eStateGet := stSDS.eTransferArmRStateGet,
    stMotionStage := stSDS.stTransferArmRStage,
    eStateSet := stSDS.eTransferArmRStateSet,
    eEnumSet := E_SDSTransferArmRStates.PREROTATE_SAMPLE_REMOVAL,
    bError := stSDS.bError,
    sErrorMsg := stSDS.sErrorMsg,
    bArrived => stSDS.bSuccess
);
END_METHOD


METHOD PRIVATE PrerotateTransferArmForInsertion
VAR_IN_OUT
    stSDS : ST_SDS;
END_VAR

stSDS.bSuccess := FALSE;

stSDS.sStatusMsg := 'Pre-rotating to allow full rotation for screwing in sample.';

SetPositionStateWaitForArrivalQuitIfError(
    eStateGet := stSDS.eTransferArmRStateGet,
    stMotionStage := stSDS.stTransferArmRStage,
    eStateSet := stSDS.eTransferArmRStateSet,
    eEnumSet := E_SDSTransferArmRStates.PREROTATE_SAMPLE_INSERTION,
    bError := stSDS.bError,
    sErrorMsg := stSDS.sErrorMsg,
    bArrived => stSDS.bSuccess
);
END_METHOD


METHOD PRIVATE RetractGarage
VAR_IN_OUT
    stSDS : ST_SDS;
END_VAR

stSDS.bSuccess := FALSE;

stSDS.sStatusMsg := 'Retracting garage.';

SetPositionStateWaitForArrivalQuitIfError(
    eStateGet := stSDS.eGarageYStateGet,
    stMotionStage := stSDS.stGarageYStage,
    eStateSet := stSDS.eGarageYStateSet,
    eEnumSet := E_SDSGarageYStates.RETRACTED,
    bError := stSDS.bError,
    sErrorMsg := stSDS.sErrorMsg,
    bArrived => stSDS.bSuccess
);
END_METHOD


METHOD PRIVATE RotateGarageForClearance
VAR_IN_OUT
    stSDS : ST_SDS;
END_VAR

stSDS.bSuccess := FALSE;

stSDS.sStatusMsg := 'Rotating garage to prevent a collision with the transfer arm sample during movement of the garage.';

IF F_Limit(
       fVal := stSDS.stGarageRStage.Axis.NcToPlc.ActPos,
       fLLim := stSDS.fGarageRotationClearancePos - stSDS.stGarageRStage.stAxisParameters.fTargetPosControlRange,
       fHLim := stSDS.fGarageRotationClearancePos + stSDS.stGarageRStage.stAxisParameters.fTargetPosControlRange,
       bInclusive := FALSE
   ) AND NOT stSDS.stGarageRStage.bBusy THEN
   stSDS.bSuccess := TRUE;
ELSE
    stSDS.stGarageRStage.fPosition := stSDS.fGarageRotationClearancePos;
    stSDS.stGarageRStage.fVelocity := stSDS.fGarageRotationSpeed;
    stSDS.stGarageRStage.bMoveCmd := TRUE;
END_IF
END_METHOD


METHOD PRIVATE RotateGarageForClearanceManual
VAR_IN_OUT
    stSDS : ST_SDS;
END_VAR

stSDS.sStatusMsg := 'Please manually rotate the garage to 45 degrees to prevent it from colliding with the sample on the transfer arm when raising it up. Click "proceed" when complete.';
END_METHOD


METHOD PRIVATE RotateToFacePort
VAR_IN_OUT
    stSDS : ST_SDS;
END_VAR

stSDS.bSuccess := FALSE;

stSDS.sStatusMsg := 'Rotating garage so that the selected slot faces the side port.';

stSDS.eFaceState := E_SDSFaceState.FACE_SIDE_PORT;

SetPositionStateWaitForArrivalQuitIfError(
    eStateGet := stSDS.eGarageRStateGet,
    stMotionStage := stSDS.stGarageRStage,
    eStateSet := stSDS.eGarageRStateSet,
    eEnumSet := stSDS.eSelectedGarageSlot,
    bError := stSDS.bError,
    sErrorMsg := stSDS.sErrorMsg,
    bArrived => stSDS.bSuccess
);
END_METHOD


METHOD PRIVATE ScrewInHalfTurn
VAR_IN_OUT
    stSDS : ST_SDS;
END_VAR

stSDS.bSuccess := FALSE;

stSDS.sStatusMsg := 'Screwing transfer arm a half turn to catch the sample pin.';

SetPositionStateWaitForArrivalQuitIfError(
    eStateGet := stSDS.eTransferArmRStateGet,
    stMotionStage := stSDS.stTransferArmRStage,
    eStateSet := stSDS.eTransferArmRStateSet,
    eEnumSet := E_SDSTransferArmRStates.SCREW_IN_HALF_TURN,
    bError := stSDS.bError,
    sErrorMsg := stSDS.sErrorMsg,
    bArrived => stSDS.bSuccess
);
END_METHOD


METHOD PRIVATE ScrewSampleIntoDiffractometer
VAR_IN_OUT
    stSDS : ST_SDS;
END_VAR

stSDS.bSuccess := FALSE;

stSDS.sStatusMsg := 'Screwing sample into diffractometer.';

SetPositionStateWaitForArrivalQuitIfError(
    eStateGet := stSDS.eTransferArmRStateGet,
    stMotionStage := stSDS.stTransferArmRStage,
    eStateSet := stSDS.eTransferArmRStateSet,
    eEnumSet := E_SDSTransferArmRStates.SCREW_INTO_DIFF,
    bError := stSDS.bError,
    sErrorMsg := stSDS.sErrorMsg,
    bArrived => stSDS.bSuccess
);
END_METHOD


METHOD PRIVATE ScrewSampleIntoGarage
VAR_IN_OUT
    stSDS : ST_SDS;
END_VAR

stSDS.bSuccess := FALSE;

stSDS.sStatusMsg := 'Screwing sample into garage.';

SetPositionStateWaitForArrivalQuitIfError(
    eStateGet := stSDS.eTransferArmRStateGet,
    stMotionStage := stSDS.stTransferArmRStage,
    eStateSet := stSDS.eTransferArmRStateSet,
    eEnumSet := E_SDSTransferArmRStates.SCREW_INTO_GARAGE,
    bError := stSDS.bError,
    sErrorMsg := stSDS.sErrorMsg,
    bArrived => stSDS.bSuccess
);
END_METHOD


METHOD PRIVATE SelectDesiredAction
VAR_INPUT
    stSDS : ST_SDS;
END_VAR

stSDS.sStatusMsg := 'Please select the desired action.';
END_METHOD


METHOD PRIVATE SelectGarageSlotForLoading
VAR_IN_OUT
    stSDS : ST_SDS;
    stSDSP : ST_SDSPersistent;
END_VAR

stSDS.sStatusMsg := 'Please select a valid garage slot to load a sample to and then click "proceed".';

IF stSDS.stUISelect.eGarageSlot >= E_SDSGarageYStates.T1 AND stSDS.stUISelect.eGarageSlot <= E_SDSGarageYStates.B4 THEN
    CASE stSDSP.astGarageSlot[stSDS.stUISelect.eGarageSlot].eState OF
        E_SampleSlotStates.DISABLED:
            stSDS.sErrorMsg := 'The selected garage slot is currently disabled.';
        E_SampleSlotStates.EMPTY:
            stSDS.eSelectedGarageSlot := stSDS.stUISelect.eGarageSlot;
        E_SampleSlotStates.FULL:
            stSDS.sErrorMsg := 'The selected garage slot is currently full.';
    END_CASE
ELSE
    stSDS.sErrorMsg := 'Please select a valid slot from T1 to B4.';
END_IF
END_METHOD


METHOD PRIVATE SelectGarageSlotForRemoval
VAR_IN_OUT
    stSDS : ST_SDS;
    stSDSP : ST_SDSPersistent;
END_VAR

stSDS.sStatusMsg := 'Please select a valid garage slot to retrieve a sample from and then click "proceed".';

IF stSDS.stUISelect.eGarageSlot >= E_SDSGarageYStates.T1 AND stSDS.stUISelect.eGarageSlot <= E_SDSGarageYStates.B4 THEN
    CASE stSDSP.astGarageSlot[stSDS.stUISelect.eGarageSlot].eState OF
        E_SampleSlotStates.DISABLED:
            stSDS.sErrorMsg := 'The selected garage slot is currently disabled.';
        E_SampleSlotStates.EMPTY:
            stSDS.sErrorMsg := 'The selected garage slot is currently empty.';
        E_SampleSlotStates.FULL:
            stSDS.eSelectedGarageSlot := stSDS.stUISelect.eGarageSlot;
    END_CASE
ELSE
    stSDS.sErrorMsg := 'Please select a valid slot from T1 to B4.';
END_IF
END_METHOD


METHOD PRIVATE SelectLoadUnloadGarage
VAR_IN_OUT
    stSDS : ST_SDS;
END_VAR

stSDS.sStatusMsg := 'Select whether you would like to load a sample to the garage or remove a sample to the garage.';

stSDS.bLoadingSelected := FALSE;
stSDS.bUnloadingSelected := FALSE;

IF stSDS.stUISelect.bLoad THEN
    stSDS.bLoadingSelected := TRUE;
ELSIF stSDS.stUISelect.bUnload THEN
    stSDS.bUnloadingSelected := TRUE;
END_IF
END_METHOD


METHOD PRIVATE SetPositionStateWaitForArrivalQuitIfError
VAR_IN_OUT
    eStateGet : UINT;
    stMotionStage : ST_MotionStage;
    eStateSet : UINT;
    bError : BOOL;
    sErrorMsg : T_MaxString;
END_VAR
VAR_INPUT
    eEnumSet : UINT;
END_VAR
VAR_OUTPUT
    bArrived : BOOL;
END_VAR

IF eStateGet = eEnumSet AND
    NOT stMotionStage.bBusy THEN
    bArrived := TRUE;
ELSIF stMotionStage.bError THEN
    bError := TRUE;
    sErrorMsg := 'And axis error occurred. Aborting sequence.';
END_IF

IF eStateGet <> eEnumSet THEN
    eStateSet := eEnumSet;
END_IF
END_METHOD


METHOD PRIVATE SetSeqState
VAR_INPUT
    stSDS : ST_SDS;
    eSeqState : E_SDSState;
END_VAR

stSDS.eSeqState := eSeqState;
END_METHOD


METHOD PRIVATE SetState
VAR_INPUT
    stSDS : ST_SDS;
    eState : E_SDSState;
END_VAR

stSDS.eState := eState;
END_METHOD


METHOD PRIVATE SetSubstate
VAR_INPUT
    stSDS : ST_SDS;
    eSubState : E_SDSState;
END_VAR

stSDS.eSubState := eSubState;
END_METHOD


METHOD PRIVATE StateMachine
VAR_IN_OUT
    stSDS : ST_SDS;
    stSDSP : ST_SDSPersistent;
END_VAR

//IF stSDS.bError THEN
//    stSDS.eState := E_SDSState.Error;
//END_IF

IF stSDS.stUISelect.bCancel THEN
    stSDS.eState := E_SDSState.Standby;
    stSDS.eSubState := E_SDSSubState.Inactive;
    stSDS.eSeqState := E_SDSSeqState.Inactive;
    stSDS.bError := FALSE;
    stSDS.sErrorMsg := '';
END_IF

stSDS.sStatusMsg := '';

CASE stSDS.eState OF
    E_SDSState.Standby:
        IF stSDS.bEnable THEN
            stSDS.eState := E_SDSState.Operating;
            stSDS.eSubState := E_SDSSubstate.Select_Desired_Action;
            stSDS.eSeqState := E_SDSSeqState.Inactive;
        ELSE
            stSDS.eSubState := E_SDSSubState.Inactive;
            stSDS.eSeqState := E_SDSSeqState.Inactive;
        END_IF
    E_SDSState.Operating:
        IF NOT stSDS.bEnable THEN
            stSDS.eState := E_SDSState.Standby;
        ELSE
            SubStateMachine(
                stSDS := stSDS,
                stSDSP := stSDSP
            );
        END_IF
    E_SDSState.Error:
        IF NOT stSDS.bError THEN
            stSDS.eState := E_SDSState.Standby;
        END_IF
        stSDS.eSubState := E_SDSSubState.Inactive;
        stSDS.eSeqState := E_SDSSeqState.Inactive;
END_CASE
END_METHOD


METHOD PRIVATE SubStateMachine
VAR_IN_OUT
    stSDS : ST_SDS;
    stSDSP : ST_SDSPersistent;
END_VAR

stSDS.bSuccess := FALSE;

CASE stSDS.eSubState OF
    E_SDSSubState.Inactive:
        ; // Do nothing
    E_SDSSubState.Select_Desired_Action:
        IF stSDS.stUISelect.bHomeGarage THEN
            stSDS.eSubState := E_SDSSubstate.Check_Can_Home_Garage;
        ELSIF stSDS.stUISelect.bHomeTransferArm THEN
            stSDS.eSubState := E_SDSSubstate.Check_Can_Home_Transfer_Arm;
        ELSIF stSDS.stUISelect.bLoadArmFromGarage THEN
            stSDS.eSubState := E_SDSSubstate.Check_Can_Load_Arm_from_Garage;
        ELSIF stSDS.stUISelect.bUnloadArmToGarage THEN
            stSDS.eSubState := E_SDSSubstate.Check_Can_Unload_Arm_to_Garage;
        ELSIF stSDS.stUISelect.bLoadUnloadGarageFromPort THEN
            stSDS.eSubState := E_SDSSubstate.Check_Can_Load_Unload_Garage_from_Port;
        ELSIF stSDS.stUISelect.bLoadDiffractometerFromArm THEN
            stSDS.eSubState := E_SDSSubstate.Check_Can_Load_Diffractometer_from_Arm;
        ELSIF stSDS.stUISelect.bUnloadDiffractometerToArm THEN
            stSDS.eSubState := E_SDSSubstate.Check_Can_Unload_Diffractometer_to_Arm;
        ELSIF stSDS.stUISelect.bManualControl THEN
            stSDS.eSubState := E_SDSSubstate.Check_Can_Manual_Control;
        END_IF
    E_SDSSubState.Check_Can_Home_Garage:
        CheckCanHomeGarage(
            stSDS := stSDS,
            stSDSP := stSDSP
        );
        IF stSDS.bSuccess THEN
            stSDS.bSuccess := FALSE;
            stSDS.eSubState := E_SDSSubstate.Home_Garage;
        END_IF
    E_SDSSubState.Home_Garage:
        HomeGarage(
            stSDS := stSDS
        );
        IF stSDS.bSuccess THEN
            stSDS.bSuccess := FALSE;
            stSDS.eState := E_SDSState.Standby;
        END_IF
    E_SDSSubState.Check_Can_Home_Transfer_Arm:
        CheckCanHomeTransferArm(
            stSDS := stSDS,
            stSDSP := stSDSP
        );
        IF stSDS.bSuccess THEN
            stSDS.bSuccess := FALSE;
            stSDS.eSubState := E_SDSSubstate.Home_Transfer_Arm;
        END_IF
    E_SDSSubState.Home_Transfer_Arm:
        HomeTransferArm(
            stSDS := stSDS
        );
        IF stSDS.bSuccess THEN
            stSDS.bSuccess := FALSE;
            stSDS.eState := E_SDSstate.Standby;
        END_IF
    E_SDSSubState.Check_Can_Load_Arm_From_Garage:
        CheckCanLoadArmFromGarage(
            stSDS := stSDS,
            stSDSP := stSDSP
        );
        IF stSDS.bSuccess THEN
            stSDS.bSuccess := FALSE;
            stSDS.eSubState := E_SDSSubstate.Load_Arm_from_Garage;
        END_IF
    E_SDSSubState.Load_Arm_from_Garage:
        LoadArmFromGarage(
            stSDS := stSDS,
            stSDSP := stSDSP
        );
        IF stSDS.bSuccess THEN
            stSDS.bSuccess := FALSE;
            stSDS.eState := E_SDSstate.Standby;
        END_IF
    E_SDSSubState.Check_Can_Load_Diffractometer_from_Arm:
        CheckCanLoadDiffractometerFromArm(
            stSDS := stSDS,
            stSDSP := stSDSP
        );
        IF stSDS.bSuccess THEN
            stSDS.bSuccess := FALSE;
            stSDS.eSubState := E_SDSSubstate.Load_Diffractometer_from_Arm;
        END_IF
    E_SDSSubState.Load_Diffractometer_from_Arm:
        LoadDiffractometerFromArm(
            stSDS := stSDS,
            stSDSP := stSDSP
        );
        IF stSDS.bSuccess THEN
            stSDS.bSuccess := FALSE;
            stSDS.eState := E_SDSstate.Standby;
        END_IF
    E_SDSSubState.Check_Can_Load_Unload_Garage_from_Port:
        CheckCanLoadUnloadGarageFromPort(
            stSDS := stSDS,
            stSDSP := stSDSP
        );
        IF stSDS.bSuccess THEN
            stSDS.bSuccess := FALSE;
            stSDS.eSubState := E_SDSSubstate.Load_Unload_Garage_from_Port;
        END_IF
    E_SDSSubState.Load_Unload_Garage_from_Port:
        LoadUnloadGarageFromPort(
            stSDS := stSDS,
            stSDSP := stSDSP
        );
        IF stSDS.bSuccess THEN
            stSDS.bSuccess := FALSE;
            stSDS.eState := E_SDSstate.Standby;
        END_IF
    E_SDSSubState.Check_Can_Unload_Arm_to_Garage:
        CheckCanUnloadArmToGarage(
            stSDS := stSDS,
            stSDSP := stSDSP
        );
        IF stSDS.bSuccess THEN
            stSDS.bSuccess := FALSE;
            stSDS.eSubState := E_SDSSubstate.Unload_Arm_to_Garage;
        END_IF
    E_SDSSubState.Unload_Arm_to_Garage:
        UnloadArmToGarage(
            stSDS := stSDS,
            stSDSP := stSDSP
        );
        IF stSDS.bSuccess THEN
            stSDS.bSuccess := FALSE;
            stSDS.eState := E_SDSstate.Standby;
        END_IF
    E_SDSSubState.Check_Can_Unload_Diffractometer_to_Arm:
        CheckCanUnloadDiffractometerToArm(
            stSDS := stSDS,
            stSDSP := stSDSP
        );
        IF stSDS.bSuccess THEN
            stSDS.bSuccess := FALSE;
            stSDS.eSubState := E_SDSSubstate.Unload_Diffractometer_to_Arm;
        END_IF
    E_SDSSubState.Unload_Diffractometer_to_Arm:
        UnloadDiffractometerToArm(
            stSDS := stSDS,
            stSDSP := stSDSP
        );
        IF stSDS.bSuccess THEN
            stSDS.bSuccess := FALSE;
            stSDS.eState := E_SDSstate.Standby;
        END_IF
    E_SDSSubState.Check_Can_Manual_Control:
        CheckCanManualControl(
            stSDS := stSDS,
            stSDSP := stSDSP
        );
        IF stSDS.bSuccess THEN
            stSDS.bSuccess := FALSE;
            stSDS.eSubState := E_SDSSubstate.Manual_Control;
        END_IF
    E_SDSSubState.Manual_Control:
        ManualControl(
            stSDS := stSDS,
            stSDSP := stSDSP
        );
        IF stSDS.bSuccess THEN
            stSDS.bSuccess := FALSE;
            stSDS.eState := E_SDSstate.Standby;
        END_IF
END_CASE
END_METHOD


METHOD PRIVATE UnloadArmToGarage
VAR_IN_OUT
    stSDS : ST_SDS;
    stSDSP : ST_SDSPersistent;
END_VAR

stSDS.bSuccess := FALSE;

CASE stSDS.eSeqState OF
    E_SDSSeqState.Inactive:
        stSDS.eSeqState := E_SDSSeqState.Home_Transfer_Arm;
    E_SDSSeqState.Home_Transfer_Arm:
        HomeTransferArm(
            stSDS := stSDS
        );
        IF stSDS.bSuccess THEN
            stSDS.bSuccess := FALSE;
            stSDS.eSeqState := E_SDSSeqState.Check_Garage_Height;
        END_IF
    E_SDSSeqState.Check_Garage_Height:
        IF stSDS.bGarageAboveCollisionHeight THEN
            stSDS.eSeqState := E_SDSSeqState.Home_Garage;
        ELSE
            stSDS.eSeqState := E_SDSSeqState.Manually_Rotate_Garage_for_Clearance_to_Raise;
        END_IF
    E_SDSSeqState.Manually_Rotate_Garage_for_Clearance_to_Raise:
        RotateGarageForClearanceManual(
            stSDS := stSDS
        );
        IF stSDS.stUISelect.bProceed THEN
            stSDS.stUISelect.bProceed := FALSE;
            stSDS.eSeqState := E_SDSSeqState.Retract_Garage_1;
        END_IF
    E_SDSSeqState.Retract_Garage_1:
        RetractGarage(
            stSDS := stSDS
        );
        IF stSDS.bSuccess THEN
            stSDS.eSeqState := E_SDSSeqState.Home_Garage;
        END_IF
    E_SDSSeqState.Home_Garage:
        HomeGarage(
            stSDS := stSDS
        );
        IF stSDS.bSuccess THEN
            stSDS.eSeqState := E_SDSSeqState.Select_Garage_Slot_for_Loading;
        END_IF
    E_SDSSeqState.Select_Garage_Slot_for_Loading:
        SelectGarageSlotForLoading(
            stSDS := stSDS,
            stSDSP := stSDSP
        );
        IF stSDS.bSuccess THEN
            stSDS.eSeqState := E_SDSSeqState.Garage_Face_Transfer_Arm;
        END_IF
    E_SDSSeqState.Garage_Face_Transfer_Arm:
        GarageFaceTransferArm(
            stSDS := stSDS
        );
        IF stSDS.bSuccess THEN
            stSDS.eSeqState := E_SDSSeqState.Rotate_Garage_for_Clearance_to_Lower;
        END_IF
    E_SDSSeqState.Rotate_Garage_for_Clearance_to_Lower:
        RotateGarageForClearance(
            stSDS := stSDS
        );
        IF stSDS.bSuccess THEN
            stSDS.eSeqState := E_SDSSeqState.Move_Garage_to_Slot_Height;
        END_IF
    E_SDSSeqState.Move_Garage_to_Slot_Height:
        MoveGarageToSlotHeight(
            stSDS := stSDS
        );
        IF stSDS.bSuccess THEN
            stSDS.eSeqState := E_SDSSeqState.Extend_Transfer_Arm_for_Insertion;
        END_IF
    E_SDSSeqState.Extend_Transfer_Arm_for_Insertion:
        ExtendTransferArmForInsertion(
            stSDS := stSDS
        );
        IF stSDS.bSuccess THEN
            stSDS.eSeqState := E_SDSSeqState.Fine_Adjustment;
        END_IF
    E_SDSSeqState.Fine_Adjustment:
        FineAdjustment(
            stSDS := stSDS
        );
        IF stSDS.stUISelect.bProceed THEN
            stSDS.eSeqState := E_SDSSeqState.Screw_Sample_into_Garage;
        END_IF
    E_SDSSeqState.Screw_Sample_into_Garage:
        ScrewSampleIntoGarage(
            stSDS := stSDS
        );
        IF stSDS.bSuccess THEN
            stSDS.eSeqState := E_SDSSeqState.Confirm_Insertion;
        END_IF
    E_SDSSeqState.Confirm_Insertion:
        ConfirmInsertion(
            stSDS := stSDS
        );
        IF stSDS.bSuccess AND stSDS.stUISelect.bProceed THEN
            stSDS.eSeqState := E_SDSSeqState.Update_Sample_Database;
        ELSIF stSDS.stUISelect.bRetry THEN
            stSDS.eSeqState := E_SDSSeqState.Fine_Adjustment;
        END_IF
    E_SDSSeqState.Update_Sample_Database:
        UpdateSampleLocationDatabaseGarageToArm(
            stSDS := stSDS,
            stSDSP := stSDSP
        );
        IF stSDS.bSuccess OR stSDS.stUISelect.bProceed THEN
            stSDS.eSeqState := E_SDSSeqState.Retract_Transfer_Arm;
        END_IF
    E_SDSSeqState.Retract_Transfer_Arm:
        HomeTransferArm(
            stSDS := stSDS
        );
        IF stSDS.bSuccess THEN
            stSDS.eSeqState := E_SDSSeqState.Rotate_Garage_for_Clearance_to_Raise;
        END_IF
    E_SDSSeqState.Rotate_Garage_for_Clearance_to_Raise:
        RotateGarageForClearance(
            stSDS := stSDS
        );
        IF stSDS.bSuccess THEN
            stSDS.eSeqState := E_SDSSeqState.Retract_Garage_2;
        END_IF
    E_SDSSeqState.Retract_Garage_2:
        RetractGarage(
            stSDS := stSDS
        );
        IF stSDS.bSuccess THEN
            stSDS.eSeqState := E_SDSSeqState.Return_Garage_to_Home;
        END_IF
    E_SDSSeqState.Return_Garage_to_Home:
        HomeGarage(
            stSDS := stSDS
        );
        IF stSDS.bSuccess THEN
            stSDS.eState := E_SDSState.Standby;
        END_IF
END_CASE
END_METHOD


METHOD PRIVATE UnloadDiffractometerToArm
VAR_IN_OUT
    stSDS : ST_SDS;
    stSDSP : ST_SDSPersistent;
END_VAR

CASE stSDS.eSeqState OF
    E_SDSSeqState.Inactive:
        stSDS.eSeqState := E_SDSSeqState.Home_Transfer_Arm;
    E_SDSSeqState.Home_Transfer_Arm:
        HomeTransferArm(
            stSDS := stSDS
        );
        IF stSDS.bSuccess THEN
            stSDS.eSeqState := E_SDSSeqState.Check_Garage_Height;
        END_IF
    E_SDSSeqState.Check_Garage_Height:
        IF stSDS.bGarageAboveCollisionHeight THEN
            stSDS.eSeqState := E_SDSSeqState.Home_Garage;
        ELSE
            stSDS.eSeqState := E_SDSSeqState.Manually_Rotate_Garage_for_Clearance_to_Raise;
        END_IF
    E_SDSSeqState.Manually_Rotate_Garage_for_Clearance_to_Raise:
        RotateGarageForClearanceManual(
            stSDS := stSDS
        );
        IF stSDS.stUISelect.bProceed THEN
            stSDS.eSeqState := E_SDSSeqState.Retract_Garage_1;
        END_IF
    E_SDSSeqState.Retract_Garage_1:
        RetractGarage(
            stSDS := stSDS
        );
        IF stSDS.bSuccess THEN
            stSDS.eSeqState := E_SDSSeqState.Home_Garage;
        END_IF
    E_SDSSeqState.Home_Garage:
        HomeGarage(
            stSDS := stSDS
        );
        IF stSDS.bSuccess THEN
            stSDS.eSeqState := E_SDSSeqState.Move_Diffractometer_to_Load_Unload_Position;
        END_IF
    E_SDSSeqState.Move_Diffractometer_to_Load_Unload_Position:
        MoveDiffractometerToLoadUnloadPosition(
            stSDS := stSDS
        );
        IF stSDS.bSuccess THEN
            stSDS.eSeqState := E_SDSSeqState.Confirm_Vacuum_Valve_Open;
        END_IF
    E_SDSSeqState.Confirm_Vacuum_Valve_Open:
        ConfirmVacuumValveOpen(
            stSDS := stSDS
        );
        IF stSDS.bSuccess THEN
            stSDS.eSeqState := E_SDSSeqState.Prerotate_Transfer_Arm_for_Extraction;
        END_IF
    E_SDSSeqState.Prerotate_Transfer_Arm_for_Extraction:
        PrerotateTransferArmForExtraction(
            stSDS := stSDS
        );
        IF stSDS.bSuccess THEN
            stSDS.eSeqState := E_SDSSeqState.Extend_Transfer_Arm_for_Diffractometer_Extraction;
        END_IF
    E_SDSSeqState.Extend_Transfer_Arm_for_Diffractometer_Extraction:
        ExtendTransferArmForDiffractometerExtraction(
            stSDS := stSDS
        );
        IF stSDS.bSuccess THEN
            stSDS.eSeqState := E_SDSSeqState.Fine_Adjustment;
        END_IF
    E_SDSSeqState.Fine_Adjustment:
        FineAdjustment(
            stSDS := stSDS
        );
        IF stSDS.stUISelect.bProceed THEN
            stSDS.eSeqState := E_SDSSeqState.Unscrew_Sample_from_Diffractometer;
        END_IF
    E_SDSSeqState.Unscrew_Sample_from_Diffractometer:
        UnscrewSampleFromDiffractometer(
            stSDS := stSDS
        );
        IF stSDS.bSuccess THEN
            stSDS.eSeqState := E_SDSSeqState.Confirm_Diffractometer_Extraction;
        END_IF
    E_SDSSeqState.Confirm_Diffractometer_Extraction:
        ConfirmDiffractometerExtraction(
            stSDS := stSDS
        );
        IF stSDS.bSuccess AND stSDS.stUISelect.bProceed THEN
            stSDS.eSeqState := E_SDSSeqState.Update_Sample_Database;
        ELSIF stSDS.stUISelect.bRetry THEN
            stSDS.eSeqState := E_SDSSeqState.Fine_Adjustment;
        END_IF
    E_SDSSeqState.Update_Sample_Database:
        UpdateSampleLocationDatabaseDiffToArm(
            stSDS := stSDS,
            stSDSP := stSDSP
        );
        IF stSDS.bSuccess OR stSDS.stUISelect.bProceed THEN
            stSDS.eSeqState := E_SDSSeqState.Retract_Transfer_Arm;
        END_IF
    E_SDSSeqState.Retract_Transfer_Arm:
        HomeTransferArm(
            stSDS := stSDS
        );
        IF stSDS.bSuccess THEN
            stSDS.eSeqState := E_SDSSeqState.Rotate_Garage_for_Clearance_to_Raise;
        END_IF
END_CASE
END_METHOD


METHOD PRIVATE UnscrewSampleFromDiffractometer
VAR_IN_OUT
    stSDS : ST_SDS;
END_VAR

stSDS.bSuccess := FALSE;

stSDS.sStatusMsg := 'Unscrewing sample from diffractometer.';

SetPositionStateWaitForArrivalQuitIfError(
    eStateGet := stSDS.eTransferArmRStateGet,
    stMotionStage := stSDS.stTransferArmRStage,
    eStateSet := stSDS.eTransferArmRStateSet,
    eEnumSet := E_SDSTransferArmRStates.UNSCREW_FROM_DIFF,
    bError := stSDS.bError,
    sErrorMsg := stSDS.sErrorMsg,
    bArrived => stSDS.bSuccess
);
END_METHOD


METHOD PRIVATE UnscrewSampleFromGarage
VAR_IN_OUT
    stSDS : ST_SDS;
END_VAR

stSDS.bSuccess := FALSE;

stSDS.sStatusMsg := 'Unscrewing sample from garage.';

SetPositionStateWaitForArrivalQuitIfError(
    eStateGet := stSDS.eTransferArmRStateGet,
    stMotionStage := stSDS.stTransferArmRStage,
    eStateSet := stSDS.eTransferArmRStateSet,
    eEnumSet := E_SDSTransferArmRStates.UNSCREW_FROM_GARAGE,
    bError := stSDS.bError,
    sErrorMsg := stSDS.sErrorMsg,
    bArrived => stSDS.bSuccess
);
END_METHOD


METHOD PRIVATE UpdateLoadUnloadAbleStatuses
VAR_IN_OUT
    stSDS : ST_SDS;
    stSDSP : ST_SDSPersistent;
END_VAR

// Determine whether the transfer arm is loadable or unloadable.
// If the transfer arm is disabled, then nothing is allowed.
// If the transfer arm is empty, it can be loaded.
// If the transfer arm is full, it can be unloaded.
CASE stSDSP.stTransferArmSlot.eState OF
    E_SampleSlotStates.EMPTY:
        stSDS.bTransferArmLoadable   := TRUE;
        stSDS.bTransferArmUnloadable := FALSE;
    E_SampleSlotStates.FULL:
        stSDS.bTransferArmLoadable   := FALSE;
        stSDS.bTransferArmUnloadable := TRUE;
    E_SampleSlotStates.DISABLED:
        stSDS.bTransferArmLoadable   := FALSE;
        stSDS.bTransferArmUnloadable := FALSE;
END_CASE

// Determine whether the diffractometer slot is loadable or unloadable.
// If the diffractometer slot is disabled, then nothing is allowed.
// If the diffractometer slot is empty, it can be loaded.
// If the diffractometer slot is full, it can be unloaded.
CASE stSDSP.stDiffractometerSlot.eState OF
    E_SampleSlotStates.EMPTY:
        stSDS.bDiffractometerLoadable   := TRUE;
        stSDS.bDiffractometerUnloadable := FALSE;
    E_SampleSlotStates.FULL:
        stSDS.bDiffractometerLoadable   := FALSE;
        stSDS.bDiffractometerUnloadable := TRUE;
    E_SampleSlotStates.DISABLED:
        stSDS.bDiffractometerLoadable   := FALSE;
        stSDS.bDiffractometerUnloadable := FALSE;
END_CASE

// Determine whether the garage is loadable or unloadable.
// If all slots in the garage are disabled, then nothing is allowed.
// If at least one slot in the garage is empty, it can be loaded.
// If at least one slot in the garage is full, it can be unloaded.
stSDS.bGarageLoadable := FALSE;
stSDS.bGarageUnloadable := FALSE;
FOR nIndex := 0 TO stSDS.nGarageSlots - 1 BY 1 DO
    CASE stSDSP.astGarageSlot[nIndex].eState OF
        E_SampleSlotStates.EMPTY:
            stSDS.bGarageLoadable   := TRUE;
        E_SampleSlotStates.FULL:
            stSDS.bGarageUnloadable := TRUE;
        E_SampleSlotStates.DISABLED:
            stSDS.bGarageLoadable := FALSE;
            stSDS.bGarageUnloadable := FALSE;
    END_CASE
END_FOR
END_METHOD


METHOD PRIVATE UpdatePositionStates
VAR_IN_OUT
    stSDS : ST_SDS;
    stSDSP : ST_SDSPersistent;
END_VAR

// Update parameters for transfer arm states.
// Horizontal axis states
fbStateSetup(stPositionState:=stSDS.astTransferArmHPosState[E_SDSTransferArmHStates.RETRACTED], sName:='RETRACTED',
    fPosition:=0,
    fVelocity:=2,
    fDelta := 2.5
);
fbStateSetup(stPositionState:=stSDS.astTransferArmHPosState[E_SDSTransferArmHStates.GARAGE_SAMPLE_REMOVAL], sName:='GARAGE_SAMPLE_REMOVAL',
    fPosition:=28,
    fVelocity:=2
);
fbStateSetup(stPositionState:=stSDS.astTransferArmHPosState[E_SDSTransferArmHStates.CONFIRM_GARAGE_EXTRACTION], sName:='CONFIRM_GARAGE_EXTRACTION',
    fPosition:=23,
    fVelocity:=2
);
fbStateSetup(stPositionState:=stSDS.astTransferArmHPosState[E_SDSTransferArmHStates.GARAGE_SAMPLE_INSERTION], sName:='GARAGE_SAMPLE_INSERTION',
    fPosition:=30,
    fVelocity:=2
);
fbStateSetup(stPositionState:=stSDS.astTransferArmHPosState[E_SDSTransferArmHStates.CONFIRM_GARAGE_INSERTION], sName:='CONFIRM_GARAGE_INSERTION',
    fPosition:=25,
    fVelocity:=2
);
fbStateSetup(stPositionState:=stSDS.astTransferArmHPosState[E_SDSTransferArmHStates.DIFF_SAMPLE_INSERTION], sName:='DIFF_SAMPLE_INSERTION',
    fPosition:=100,
    fVelocity:=2
);
fbStateSetup(stPositionState:=stSDS.astTransferArmHPosState[E_SDSTransferArmHStates.DIFF_SAMPLE_EXTRACTION], sName:='DIFF_SAMPLE_EXTRACTION',
    fPosition:=100,
    fVelocity:=2
);
fbStateSetup(stPositionState:=stSDS.astTransferArmHPosState[E_SDSTransferArmHStates.CONFIRM_DIFF_INSERTION], sName:='CONFIRM_DIFF_INSERTION',
    fPosition:=75,
    fVelocity:=2
);
fbStateSetup(stPositionState:=stSDS.astTransferArmHPosState[E_SDSTransferArmHStates.CONFIRM_DIFF_EXTRACTION], sName:='CONFIRM_DIFF_EXTRACTION',
    fPosition:=75,
    fVelocity:=2
);

// Rotational axis states
fbStateSetup(stPositionState:=stSDS.astTransferArmRPosState[E_SDSTransferArmRStates.FULLY_CCW], sName:='FULLY_CCW',
    fPosition:=0,
    fVelocity:=stSDS.fGarageRotationSpeed,
    fDelta := 5.0
);
IF NOT stSDS.stTransferArmRStage.bLimitForwardEnable THEN
    fbStateSetup(stPositionState:=stSDS.astTransferArmRPosState[E_SDSTransferArmRStates.PREROTATE_SAMPLE_REMOVAL], sName:='PREROTATE_SAMPLE_REMOVAL',
        fPosition:=stSDS.stTransferArmRStage.Axis.NcToPlc.ActPos,
        fVelocity:=stSDS.fTransferArmRotationSpeed
    );
ELSE
    fbStateSetup(stPositionState:=stSDS.astTransferArmRPosState[E_SDSTransferArmRStates.PREROTATE_SAMPLE_REMOVAL], sName:='PREROTATE_SAMPLE_REMOVAL',
        fPosition:=20000,
        fVelocity:=stSDS.fTransferArmRotationSpeed
    );
END_IF
IF NOT stSDS.stTransferArmRStage.bLimitBackwardEnable THEN
    fbStateSetup(stPositionState:=stSDS.astTransferArmRPosState[E_SDSTransferArmRStates.PREROTATE_SAMPLE_INSERTION], sName:='PREROTATE_SAMPLE_INSERTION',
        fPosition:=stSDS.stTransferArmRStage.Axis.NcToPlc.ActPos,
        fVelocity:=stSDS.fTransferArmRotationSpeed
    );
ELSE
    fbStateSetup(stPositionState:=stSDS.astTransferArmRPosState[E_SDSTransferArmRStates.PREROTATE_SAMPLE_INSERTION], sName:='PREROTATE_SAMPLE_INSERTION',
        fPosition:=-20000,
        fVelocity:=stSDS.fTransferArmRotationSpeed
    );
END_IF
fbStateSetup(stPositionState:=stSDS.astTransferArmRPosState[E_SDSTransferArmRStates.UNSCREW_FROM_GARAGE], sName:='UNSCREW_FROM_GARAGE',
    fPosition:=0,
    fVelocity:=stSDS.fTransferArmRotationSpeed
);
fbStateSetup(stPositionState:=stSDS.astTransferArmRPosState[E_SDSTransferArmRStates.UNSCREW_FROM_DIFF], sName:='UNSCREW_FROM_DIFF',
    fPosition:=0,
    fVelocity:=stSDS.fTransferArmRotationSpeed
);
fbStateSetup(stPositionState:=stSDS.astTransferArmRPosState[E_SDSTransferArmRStates.SCREW_INTO_GARAGE], sName:='SCREW_INTO_GARAGE',
    fPosition:=1700,
    fVelocity:=stSDS.fTransferArmRotationSpeed
);
fbStateSetup(stPositionState:=stSDS.astTransferArmRPosState[E_SDSTransferArmRStates.SCREW_INTO_DIFF], sName:='SCREW_INTO_DIFF',
    fPosition:=1700,
    fVelocity:=stSDS.fTransferArmRotationSpeed
);
fbStateSetup(stPositionState:=stSDS.astTransferArmRPosState[E_SDSTransferArmRStates.SCREW_IN_HALF_TURN], sName:='SCREW_IN_HALF_TURN',
    fPosition:=stSDS.stTransferArmRStage.Axis.NcToPlc.ActPos + 180,
    fVelocity:=stSDS.fTransferArmRotationSpeed
);

// Update parameters for garage states.
// Y axis states
fbStateSetup(
    stPositionState := stSDS.astGarageYPosState[E_SDSGarageYStates.RETRACTED], sName:='RETRACTED',
    fPosition := 0.0,
    fVelocity := 1.0,
    fDelta := 10.0
);

FOR nIndex := E_SDSGarageYStates.T1 TO E_SDSGarageYStates.B4 BY 1 DO
    fbStateSetup(
        stPositionState := stSDS.astGarageYPosState[nIndex],
        sName := stSDSP.astGarageSlot[nIndex].sTag,
        fPosition := stSDSP.astGarageSlot[nIndex].fYPos,
        fVelocity := 1.0,
    );
END_FOR

// Rotational axis states
fbStateSetup(
    stPositionState := stSDS.astGarageRPosState[E_SDSGarageRStates.PREDICTED_HOME], sName:='PREDICTED_HOME',
    fPosition := 0.0,
    fVelocity := 10.0,
    fDelta := 1.0,
    bLocked := TRUE
);

FOR nIndex := E_SDSGarageYStates.T1 TO E_SDSGarageYStates.B4 BY 1 DO
    CASE stSDS.eFaceState OF
        E_SDSFaceState.FACE_SIDE_PORT:
            fbStateSetup(
                stPositionState := stSDS.astGarageRPosState[nIndex],
                sName := stSDSP.astGarageSlot[nIndex].sTag,
                fPosition := stSDSP.astGarageSlot[nIndex].fDeg + stSDS.fFacePortOffset,
                fVelocity := 10.0,
            );
    ELSE
        fbStateSetup(
            stPositionState := stSDS.astGarageRPosState[nIndex],
            sName := stSDSP.astGarageSlot[nIndex].sTag,
            fPosition := stSDSP.astGarageSlot[nIndex].fDeg,
            fVelocity := 10.0,
        );
    END_CASE
END_FOR
END_METHOD


METHOD PRIVATE UpdateSampleLocationDatabaseDiffToArm
VAR_IN_OUT
    stSDS : ST_SDS;
    stSDSP : ST_SDSPersistent;
END_VAR
VAR
    stTempSlot : ST_SampleSlot;
END_VAR

stSDS.bSuccess := FALSE;

stTempSlot := stSDSP.stTransferArmSlot;

stSDS.sStatusMsg := 'Updating the sample database.';

IF stSDS.eSelectedGarageSlot >= E_SDSGarageYStates.T1 AND stSDS.eSelectedGarageSlot <= E_SDSGarageYStates.B4 THEN
    stSDSP.stTransferArmSlot.eState := stSDSP.stDiffractometerSlot.eState;
    stSDSP.stTransferArmSlot.sDesc := stSDSP.stDiffractometerSlot.sDesc;

    stSDSP.stDiffractometerSlot.eState := stTempSlot.eState;
    stSDSP.stDiffractometerSlot.sDesc := stTempSlot.sDesc;

    stSDS.bSuccess := TRUE;
ELSE
    stSDS.sErrorMsg := 'Failed to automatically update sample position in database. Invalid slot selected. Sequence will continue, but please manually update the database from the interface. After manually updating the database, click "proceed" to continue.';
END_IF
END_METHOD


METHOD PRIVATE UpdateSampleLocationDatabaseGarageToArm
VAR_IN_OUT
    stSDS : ST_SDS;
    stSDSP : ST_SDSPersistent;
END_VAR
VAR
    stTempSlot : ST_SampleSlot;
END_VAR

stSDS.bSuccess := FALSE;

stTempSlot := stSDSP.stTransferArmSlot;

stSDS.sStatusMsg := 'Updating the sample database.';

IF stSDS.eSelectedGarageSlot >= E_SDSGarageYStates.T1 AND stSDS.eSelectedGarageSlot <= E_SDSGarageYStates.B4 THEN
    stSDSP.stTransferArmSlot.eState := stSDSP.astGarageSlot[stSDS.eSelectedGarageSlot].eState;
    stSDSP.stTransferArmSlot.sDesc := stSDSP.astGarageSlot[stSDS.eSelectedGarageSlot].sDesc;

    stSDSP.astGarageSlot[stSDS.eSelectedGarageSlot].eState := stTempSlot.eState;
    stSDSP.astGarageSlot[stSDS.eSelectedGarageSlot].sDesc := stTempSlot.sDesc;

    stSDS.bSuccess := TRUE;
ELSE
    stSDS.sErrorMsg := 'Failed to automatically update sample position in database. Invalid slot selected. Sequence will continue, but please manually update the database from the interface. After manually updating the database, click "proceed" to continue.';
END_IF
END_METHOD


METHOD PRIVATE UpdateSampleLocationDatabaseManualExtraction
VAR_IN_OUT
    stSDS : ST_SDS;
    stSDSP : ST_SDSPersistent;
END_VAR

stSDS.bSuccess := FALSE;

stSDS.sStatusMsg := 'Please extract the sample. Click "proceed" when you have finished.';

IF stSDS.eSelectedGarageSlot >= E_SDSGarageYStates.T1 AND stSDS.eSelectedGarageSlot <= E_SDSGarageYStates.B4 THEN
    stSDSP.astGarageSlot[stSDS.eSelectedGarageSlot].eState := E_SampleSlotStates.EMPTY;
    stSDSP.astGarageSlot[stSDS.eSelectedGarageSlot].sDesc := '';
ELSE
    stSDS.sErrorMsg := 'Failed to update sample position in database. Invalid slot selected. Sequence will continue, but please manually update the database from the interface.';
END_IF
END_METHOD


METHOD PRIVATE UpdateSampleLocationDatabaseManualInsertion
VAR_IN_OUT
    stSDS : ST_SDS;
    stSDSP : ST_SDSPersistent;
END_VAR

stSDS.bSuccess := FALSE;

stSDS.sStatusMsg := 'Please insert the sample and write an identifying description for it in the text field. Click "proceed" when you have finished.';

IF stSDS.eSelectedGarageSlot >= E_SDSGarageYStates.T1 AND stSDS.eSelectedGarageSlot <= E_SDSGarageYStates.B4 THEN
    stSDSP.astGarageSlot[stSDS.eSelectedGarageSlot].eState := E_SampleSlotStates.FULL;
    stSDSP.astGarageSlot[stSDS.eSelectedGarageSlot].sDesc := stSDS.stUISelect.sTextInput;
ELSE
    stSDS.sErrorMsg := 'Failed to update sample position in database. Invalid slot selected. Sequence will continue, but please manually update the database from the interface.';
END_IF
END_METHOD

END_FUNCTION_BLOCK

// ---- POUs/PRG_RotDet.TcPOU

PROGRAM PRG_RotDet
VAR
    fb_Rot_Det : FB_MotionStage;
    bInit : BOOl := TRUE;
END_VAR


IF ( bInit) THEN
   bInit := FALSE;
   Main.M45.bHardwareEnable := TRUE;
   Main.M45.bPowerSelf := TRUE;
   Main.M45.nBrakeMode := ENUM_StageBrakeMode.NO_BRAKE;
   Main.M45.nEnableMode := ENUM_StageEnableMode.DURING_MOTION;
   Main.M45.bLimitForwardEnable := TRUE;
   Main.M45.bLimitBackwardEnable := TRUE;
   Main.M45.fVelocity := 0.1;
END_IF

fb_Rot_Det(stMotionStage:=Main.M45);

END_PROGRAM

// ---- POUs/PRG_SpetrometerArm.TcPOU

PROGRAM PRG_SpetrometerArm
VAR
        {attribute 'TcLinkTo' := 'TIIB[Rack#1A-01 Coupler (EK1100)]^Rack#1A-02 SFIN (EL1918)^StandardOutputs^Standard In Var 2'}
    bEnaIclk AT %Q*: BOOL := TRUE;

    {attribute 'TcLinkTo' := 'TIIB[Rack#1A-01 Coupler (EK1100)]^Rack#1A-02 SFIN (EL1918)^StandardOutputs^Standard In Var 1'}
    bEnaIclkErrAck AT %Q*: BOOL := FALSE;

    {attribute 'TcLinkTo' := 'TIIB[Rack#1A-01 Coupler (EK1100)]^Rack#1A-02 SFIN (EL1918)^StandardOutputs^Standard In Var 9'}
    bEnaIclkRestartESTOP AT %Q*: BOOL := FALSE;

    fbPower_AxisM11: MC_Power;
    fbPower_AxisM12: MC_Power;
    fbPower_AxisM13: MC_Power;
    fbPower_AxisM14: MC_Power;

    rtESTOPDeactivated: R_TRIG;

    tonTurnoffCBReset: TON;
END_VAR


ACT_ESTOP();

PRG_2Theta();
PRG_DET_ARM();
PRG_DET_CHAMBER();
PRG_DET_SLIT();
PRG_DET_FRAME();
PRG_OPT_SLITS();
PRG_OPT_YG();
PRG_OPT_XPM();
PRG_OPT();
PRG_Sensor();

tonTurnOffCBReset(IN:=
    GVL_VAR.bCircuitBreakerB0108Reset OR
    GVL_VAR.bCircuitBreakerB0113Reset OR
    GVL_VAR.bCircuitBreakerB0118Reset OR
    GVL_VAR.bCircuitBreakerR2A02Reset OR
    GVL_VAR.bCircuitBreakerR2A07Reset OR
    GVL_VAR.bCircuitBreakerR2A13Reset OR
    GVL_VAR.bCircuitBreakerR2B14Reset OR
    GVL_VAR.bCircuitBreakerR2B17Reset,
    PT:=T#2s
);
IF tonTurnOffCBReset.Q THEN
    GVL_VAR.bCircuitBreakerB0108Reset := FALSE;
    GVL_VAR.bCircuitBreakerB0113Reset := FALSE;
    GVL_VAR.bCircuitBreakerB0118Reset := FALSE;
    GVL_VAR.bCircuitBreakerR2A02Reset := FALSE;
    GVL_VAR.bCircuitBreakerR2A07Reset := FALSE;
    GVL_VAR.bCircuitBreakerR2A13Reset := FALSE;
    GVL_VAR.bCircuitBreakerR2B14Reset := FALSE;
    GVL_VAR.bCircuitBreakerR2B17Reset := FALSE;
END_IF

ACTION ACT_ESTOP:

IF bEnaIclkErrAck THEN
    bEnaIclkErrAck := FALSE;
END_IF
IF bEnaIclkRestartESTOP THEN
    bEnaIclkRestartESTOP := FALSE;
END_IF

// When user push the ESTOPs
// REVALUATE AFTER TESTING:
// Only specific motors are a part of the ESTOP at this point based on
// "Components" column on this page:
// https://confluence.slac.stanford.edu/display/L2SI/qRIXS+Spectrometer+Arm
// Items are commented out if not included in ESTOP to allow them to be added back easily.
IF NOT GVL_EPS.bESTOP THEN

    GVL_EPS.bOpenSV1 := FALSE;
    GVL_EPS.bOpenSV2 := FALSE;

    Main.M1.bHardwareEnable := FALSE; // SSL Sliding Seal // QRIX:SSL:MMS
    Main.M2.bHardwareEnable := FALSE; // 2Theta Arm // QRIX:SA:MMS:2Theta
    //Main.M3.bHardwareEnable := FALSE; // Optics Slits XS1 // QRIX:OPTSL:MMS:NORTH
    //Main.M4.bHardwareEnable := FALSE; // Optics Slits XS2 // QRIX:OPTSL:MMS:SOUTH
    //Main.M5.bHardwareEnable := FALSE; // Optics Slits YS1 // QRIX:OPTSL:MMS:TOP
    //Main.M6.bHardwareEnable := FALSE; // Optics Slits YS2 // QRIX:OPTSL:MMS:BOTTOM
    Main.M7.bHardwareEnable := FALSE; // Optics Base YG1 // QRIX:OPT:MMS:Y1
    Main.M8.bHardwareEnable := FALSE; // Optics Base YG2 // QRIX:OPT:MMS:Y2
    Main.M9.bHardwareEnable := FALSE; // Optics Base YG3 // QRIX:OPT:MMS:Y3
    //Main.M10.bHardwareEnable := FALSE; // Optics Grating RxG // QRIX:G:MMS:Rx
    //Main.M11.bHardwareEnable := FALSE; // Optics Grating XG // QRIX:G:MMS:X
    //Main.M12.bHardwareEnable := FALSE; // Optics Mirror XPM1 // QRIX:PM:MMS:X1
    //Main.M13.bHardwareEnable := FALSE; // Optics Mirror XPM2 // QRIX:PM:MMS:X2
    //Main.M14.bHardwareEnable := FALSE; // Optics Mirror RzPM // QRIX:PM:MMS:Rz
    Main.M15.bHardwareEnable := FALSE; // Detector Frame YDF1 // QRIX:DF:MMS:Y1
    Main.M16.bHardwareEnable := FALSE; // Detector Frame YDF2 // QRIX:DF:MMS:Y2
    Main.M17.bHardwareEnable := FALSE; // Detector Frame YDF3 // QRIX:DF:MMS:Y3
    //Main.M18.bHardwareEnable := FALSE; // Detector Slits XSDC1 // QRIX:DETSL:MMS:NORTH
    //Main.M19.bHardwareEnable := FALSE; // Detector Slits XSDC2 // QRIX:DETSL:MMS:SOUTH
    //Main.M20.bHardwareEnable := FALSE; // Detector Slits YSDC1 // QRIX:DETSL:MMS:TOP
    //Main.M21.bHardwareEnable := FALSE; // Detector Slits YSDC2 // QRIX:DETSL:MMS:BOTTOM
    //Main.M22.bHardwareEnable := FALSE; // Detector Chamber XDC // QRIX:DC:MMS:X
    //Main.M23.bHardwareEnable := FALSE; // Detector Chamber RyDC // QRIX:DC:MMS:Ry
    //Main.M24.bHardwareEnable := FALSE; // Detector Chamber ZDC // QRIX:DC:MMS:Z
    Main.M25.bHardwareEnable := FALSE; // Detector Arm YF1 // QRIX:DA:MMS:Y1
    Main.M26.bHardwareEnable := FALSE; // Detector Arm YF2 // QRIX:DA:MMS:Y2
    Main.M27.bHardwareEnable := FALSE; // Detector Arm ZF // QRIX:DA:MMS:Z

    bDoneJackOff := FALSE;
    bDoneLevitation := FALSE;
    bDoneLanding := FALSE;
    bDoneAdjustingRoll := FALSE;
    bDoneAdjustingPitch := FALSE;
    bDoneAdjustingHeight := FALSE;
END_IF
rtESTOPDeactivated(CLK:=GVL_EPS.bESTOP);
IF rtESTOPDeactivated.Q THEN
    Main.M1.bHardwareEnable := TRUE; // SSL Sliding Seal // QRIX:SSL:MMS
    Main.M2.bHardwareEnable := TRUE; // 2Theta Arm // QRIX:SA:MMS:2Theta
    //Main.M3.bHardwareEnable := TRUE; // Optics Slits XS1 // QRIX:OPTSL:MMS:NORTH
    //Main.M4.bHardwareEnable := TRUE; // Optics Slits XS2 // QRIX:OPTSL:MMS:SOUTH
    //Main.M5.bHardwareEnable := TRUE; // Optics Slits YS1 // QRIX:OPTSL:MMS:TOP
    //Main.M6.bHardwareEnable := TRUE; // Optics Slits YS2 // QRIX:OPTSL:MMS:BOTTOM
    Main.M7.bHardwareEnable := TRUE; // Optics Base YG1 // QRIX:OPT:MMS:Y1
    Main.M8.bHardwareEnable := TRUE; // Optics Base YG2 // QRIX:OPT:MMS:Y2
    Main.M9.bHardwareEnable := TRUE; // Optics Base YG3 // QRIX:OPT:MMS:Y3
    //Main.M10.bHardwareEnable := TRUE; // Optics Grating RxG // QRIX:G:MMS:Rx
    //Main.M11.bHardwareEnable := TRUE; // Optics Grating XG // QRIX:G:MMS:X
    //Main.M12.bHardwareEnable := TRUE; // Optics Mirror XPM1 // QRIX:PM:MMS:X1
    //Main.M13.bHardwareEnable := TRUE; // Optics Mirror XPM2 // QRIX:PM:MMS:X2
    //Main.M14.bHardwareEnable := TRUE; // Optics Mirror RzPM // QRIX:PM:MMS:Rz
    Main.M15.bHardwareEnable := TRUE; // Detector Frame YDF1 // QRIX:DF:MMS:Y1
    Main.M16.bHardwareEnable := TRUE; // Detector Frame YDF2 // QRIX:DF:MMS:Y2
    Main.M17.bHardwareEnable := TRUE; // Detector Frame YDF3 // QRIX:DF:MMS:Y3
    //Main.M18.bHardwareEnable := TRUE; // Detector Slits XSDC1 // QRIX:DETSL:MMS:NORTH
    //Main.M19.bHardwareEnable := TRUE; // Detector Slits XSDC2 // QRIX:DETSL:MMS:SOUTH
    //Main.M20.bHardwareEnable := TRUE; // Detector Slits YSDC1 // QRIX:DETSL:MMS:TOP
    //Main.M21.bHardwareEnable := TRUE; // Detector Slits YSDC2 // QRIX:DETSL:MMS:BOTTOM
    //Main.M22.bHardwareEnable := TRUE; // Detector Chamber XDC // QRIX:DC:MMS:X
    //Main.M23.bHardwareEnable := TRUE; // Detector Chamber RyDC // QRIX:DC:MMS:Ry
    //Main.M24.bHardwareEnable := TRUE; // Detector Chamber ZDC // QRIX:DC:MMS:Z
    Main.M25.bHardwareEnable := TRUE; // Detector Arm YF1 // QRIX:DA:MMS:Y1
    Main.M26.bHardwareEnable := TRUE; // Detector Arm YF2 // QRIX:DA:MMS:Y2
    Main.M27.bHardwareEnable := TRUE; // Detector Arm ZF // QRIX:DA:MMS:Z
END_IF

// Disable M1(Servo) and M2(Stepper) if the frame is landing...
IF NOT GVL_Sensor.bFloating THEN
    //Main.M1.bEnable := FALSE;
    //Main.M2.bEnable := FALSE;
END_IF


// When user requests to reset ESTOP.
IF GVL_EPS.bResetIclk THEN
    GVL_EPS.bResetIclk := FALSE;
    bEnaIclkErrAck := TRUE;
    bEnaIclkRestartESTOP := TRUE;
END_IF
END_ACTION

END_PROGRAM

// ---- Spectometer Arm POUs/PRG_2Theta.TcPOU

PROGRAM PRG_2Theta
VAR
    bInit: BOOL := TRUE;
    fbPower_AxisM2:  MC_Power;
    fb2ThetaStepper : FB_MotionStage;
    bMoveOk: BOOL;
    iEnableMotorState: UINT;
    tonEnableMotorTimeout: TON;
    tEnableMotorTimeoutTime: TIME := T#5s;
    bMovePos: BOOL;
    bMoveNeg: BOOL;
    bMovePosAndOK: BOOL;
    bMoveNegAndOK: BOOL;
    rtExecuteMove: R_TRIG;

    {attribute 'TcLinkTo' :=  'TIID^Device 2 (EtherCAT)^Rack#1A-01 Coupler (EK1100)^Rack#1A-04 DR_2Th (EL7047)^STM Status^Status^Ready'}
    b2ThetaDriveReady AT %I*: BOOL;
    {attribute 'TcLinkTo' :=  'TIPC^qrix_motion^qrix_motion Instance^PlcTask Outputs^PRG_SSL.EL7047_02_01_SSL_Status_to_NC'}
    nSSLDriveStatus AT %I* : USINT;
    bSSLDriveReady : BOOL;
END_VAR

VAR CONSTANT
    fThresholdPS1: REAL := 0.15;
    fThresholdPS2: REAL := 0.15;
    fThresholdPS3: REAL := 0.15;
END_VAR


IF binit THEN
    bInit := FALSE;

    // Stepper
    //Main.M2.nBrakeMode := ENUM_StageBrakeMode.IF_ENABLED;
    // Disabled brake. It actually doesn't help with anything and we found that it
    // is sometimes interfering with the movement of the motor. We think it might be
    // some sort of lag in the brake disengaging that causes it to fight with the
    // drive for a bit, which causes overcurrent faults.
    Main.M2.nBrakeMode := ENUM_StageBrakeMode.IF_MOVING;
    Main.M2.bBrakeRelease := TRUE;
    Main.M2.bHardwareEnable := TRUE;
    Main.M2.bPowerSelf := TRUE;

    Main.M2.nEnableMode := ENUM_StageEnableMode.NEVER ;
END_IF;

bSSLDriveReady := nSSLDriveStatus.1; // Drive status ready bit after tying it to bFloating.

ACT_Stepper();

ACTION ACT_Stepper:

// Simplified enabling logic by removing separate fbPower function and
// making the estop and other permissives drive the bPowerSelf bit.
// Now, the motor motion is handled entirely within the FB_MotionStage block
// which makes this usage more standard and easier to work with using our
// standard typhos widget.
Main.M2.bHardwareEnable := 		GVL_EPS.bESTOP // ESTOP
                            AND GVL_Sensor.bFloating
                            AND	GVL_Sensor.stPS1.fValue > fThresholdPS1
                            AND GVL_Sensor.stPS2.fValue > fThresholdPS2
                            AND GVL_Sensor.stPS3.fValue > fThresholdPS3 // Compressed-air pressure
                            AND GVL_EPS.bOpenSV1
                            AND GVL_EPS.bOpenSV2;

IF NOT PRG_SSL.bRealignCouple THEN
    CASE iEnableMotorState OF
        0:
            IF Main.M2.bExecute AND GVL_Sensor.bFloating THEN
                rtExecuteMove(CLK:=FALSE);
                Main.M2.bExecute := FALSE;
                Main.M2.bEnable := TRUE;
                Main.M1.bEnable := TRUE;
                iEnableMotorState := iEnableMotorState + 1;
            ELSIF Main.M2.bExecute AND NOT GVL_Sensor.bFloating THEN
                Main.M2.bExecute := FALSE;
                Main.M2.bError := TRUE;
                Main.M1.bError := TRUE;
                Main.M2.sCustomErrorMessage := 'Move failed. Arm must be levitating to move.';
                Main.M1.sCustomErrorMessage := 'Move failed. Arm must be levitating to move.';
            ELSE
                Main.M2.bEnable := FALSE;
                Main.M1.bEnable := FALSE;
            END_IF
            tonEnableMotorTimeout(IN:=FALSE);
        1: // Wait until the logic confirms both motors are fully enabled
            tonEnableMotorTimeout(IN:=NOT Main.M2.bAllEnable OR NOT Main.M1.bAllEnable,PT:=tEnableMotorTimeoutTime);

            // Check which direction we are moving, and if the directional enables will allow that move.
            bMovePos        := Main.M2.stAxisStatus.fActPosition < Main.M2.fPosition;
            bMoveNeg        := Main.M2.stAxisStatus.fActPosition > Main.M2.fPosition;
            bMovePosAndOK   := bMovePos AND Main.M2.bAllForwardEnable AND Main.M1.bAllForwardEnable;
            bMoveNegAndOK   := bMoveNeg AND Main.M2.bAllBackwardEnable AND Main.M1.bAllBackwardEnable;

            // Check for fully enabled
            IF Main.M2.bAllEnable AND Main.M1.bAllEnable THEN
                // Check direction of motion and if that direction is enabled
                IF bMovePosAndOK OR bMoveNegAndOK THEN
                    iEnableMotorState := iEnableMotorState + 1;
                    tonEnableMotorTimeout(IN:=FALSE);
                ELSE
                    IF NOT Main.M2.bError OR Main.M1.bError THEN
                        // Direction of motion is not enabled, so let's report the error and give a helpful error message.
                        Main.M2.bError := TRUE;
                        Main.M1.bError := TRUE;
                        IF bMovePos THEN
                            IF NOT Main.M2.bLimitForwardEnable THEN
                                Main.M2.sCustomErrorMessage := 'Move forward failed due to forward limit switch.';
                                Main.M1.sCustomErrorMessage := 'Move forward failed due to forward limit switch for 2 theta motor.';
                            ELSIF NOT Main.M1.bLimitForwardEnable THEN
                                Main.M1.sCustomErrorMessage := 'Move forward failed due to forward limit switch.';
                                Main.M2.sCustomErrorMessage := 'Move forward failed due to forward limit switch for SSL motor.';
                            ELSIF NOT Main.M2.bGantryForwardEnable AND Main.M2.bGantryAxis THEN
                                Main.M2.sCustomErrorMessage := 'Move forward failed due to gantry motion tolerance limit.';
                                Main.M1.sCustomErrorMessage := 'Move forward failed due to gantry motion tolerance limit for 2 theta motor.';
                            ELSIF NOT Main.M1.bGantryForwardEnable AND Main.M1.bGantryAxis THEN
                                Main.M1.sCustomErrorMessage := 'Move forward failed due to gantry motion tolerance limit.';
                                Main.M2.sCustomErrorMessage := 'Move forward failed due to gantry motion tolerance limit for SSL motor.';
                            ELSIF NOT Main.M2.stEPSForwardEnable.bEPS_OK THEN
                                Main.M2.sCustomErrorMessage := 'Move forward failed due to EPS condition.';
                                Main.M1.sCustomErrorMessage := 'Move forward failed due to EPS condition for 2 theta motor.';
                            ELSIF NOT Main.M1.stEPSForwardEnable.bEPS_OK THEN
                                Main.M1.sCustomErrorMessage := 'Move forward failed due to EPS condition.';
                                Main.M2.sCustomErrorMessage := 'Move forward failed due to EPS condition for SSL motor.';
                            ELSE
                                Main.M1.sCustomErrorMessage := 'Move forward failed for unspecified reason.';
                                Main.M2.sCustomErrorMessage := 'Move forward failed for unspecified reason.';
                            END_IF
                        ELSIF bMoveNeg THEN
                            IF NOT Main.M2.bLimitBackwardEnable THEN
                                Main.M2.sCustomErrorMessage := 'Move backward failed due to forward limit switch.';
                                Main.M1.sCustomErrorMessage := 'Move backward failed due to forward limit switch for 2 theta motor.';
                            ELSIF NOT Main.M1.bLimitBackwardEnable THEN
                                Main.M1.sCustomErrorMessage := 'Move backward failed due to forward limit switch.';
                                Main.M2.sCustomErrorMessage := 'Move backward failed due to forward limit switch for SSL motor.';
                            ELSIF NOT Main.M2.bGantryBackwardEnable AND Main.M2.bGantryAxis THEN
                                Main.M2.sCustomErrorMessage := 'Move backward failed due to gantry motion tolerance limit.';
                                Main.M1.sCustomErrorMessage := 'Move backward failed due to gantry motion tolerance limit for 2 theta motor.';
                            ELSIF NOT Main.M1.bGantryBackwardEnable AND Main.M1.bGantryAxis THEN
                                Main.M1.sCustomErrorMessage := 'Move backward failed due to gantry motion tolerance limit.';
                                Main.M2.sCustomErrorMessage := 'Move backward failed due to gantry motion tolerance limit for SSL motor.';
                            ELSIF NOT Main.M2.stEPSBackwardEnable.bEPS_OK THEN
                                Main.M2.sCustomErrorMessage := 'Move backward failed due to EPS condition.';
                                Main.M1.sCustomErrorMessage := 'Move backward failed due to EPS condition for 2 theta motor.';
                            ELSIF NOT Main.M1.stEPSBackwardEnable.bEPS_OK THEN
                                Main.M1.sCustomErrorMessage := 'Move backward failed due to EPS condition.';
                                Main.M2.sCustomErrorMessage := 'Move backward failed due to EPS condition for SSL motor.';
                            ELSE
                                Main.M2.sCustomErrorMessage := 'Move backward failed for unspecified reason.';
                                Main.M1.sCustomErrorMessage := 'Move backward failed for unspecified reason.';
                            END_IF
                        ELSE
                            Main.M2.sCustomErrorMessage := 'Move failed because it was not large enough to register.';
                            Main.M1.sCustomErrorMessage := 'Move failed because it was not large enough to register.';
                        END_IF
                    END_IF
                    iEnableMotorState := 0;
                END_IF
            ELSIF tonEnableMotorTimeout.Q THEN
                IF NOT Main.M2.bError OR Main.M1.bError THEN
                    Main.M2.bError := TRUE;
                    Main.M1.bError := TRUE;
                    IF NOT Main.M2.bEnable THEN
                        Main.M2.sCustomErrorMessage := 'Move never enabled because bEnable never received.';
                        Main.M1.sCustomErrorMessage := 'Move never enabled because bEnable never received on 2 theta motor.';
                    ELSIF NOT Main.M1.bEnable THEN
                        Main.M1.sCustomErrorMessage := 'Move never enabled because bEnable never received.';
                        Main.M2.sCustomErrorMessage := 'Move never enabled because bEnable never received on SSL motor.';
                    ELSIF NOT Main.M2.bHardwareEnable THEN
                        Main.M2.sCustomErrorMessage := 'Move never enabled because bHardwareEnable set false.';
                        Main.M1.sCustomErrorMessage := 'Move never enabled because bHardwareEnable set false on 2 theta motor.';
                    ELSIF NOT Main.M1.bHardwareEnable THEN
                        Main.M1.sCustomErrorMessage := 'Move never enabled because bHardwareEnable set false.';
                        Main.M2.sCustomErrorMessage := 'Move never enabled because bHardwareEnable set false on SSL motor.';
                    ELSIF NOT Main.M2.stEPSPowerEnable.bEPS_OK THEN
                        Main.M2.sCustomErrorMessage := 'Move never enabled because of EPS condition.';
                        Main.M1.sCustomErrorMessage := 'Move never enabled because of EPS condition on 2 theta motor.';
                    ELSIF NOT Main.M1.stEPSPowerEnable.bEPS_OK THEN
                        Main.M1.sCustomErrorMessage := 'Move never enabled because of EPS condition.';
                        Main.M2.sCustomErrorMessage := 'Move never enabled because of EPS condition on SSL motor.';
                    ELSIF NOT Main.M2.bUserEnable THEN
                        Main.M2.sCustomErrorMessage := 'Move never enabled because user enable is set to false.';
                        Main.M1.sCustomErrorMessage := 'Move never enabled because user enable is set to false on 2 theta motor.';
                    ELSIF NOT Main.M1.bUserEnable THEN
                        Main.M1.sCustomErrorMessage := 'Move never enabled because user enable is set to false.';
                        Main.M2.sCustomErrorMessage := 'Move never enabled because user enable is set to false on SSL motor.';
                    ELSE
                        Main.M2.sCustomErrorMessage := 'Move never enabled in the timeout duration.';
                        Main.M1.sCustomErrorMessage := 'Move never enabled in the timeout duration.';
                    END_IF
                END_IF
                iEnableMotorState := 0;
            END_IF
        2: // Wait for the motor drives to switch to the ready state before commanding the move.
            tonEnableMotorTimeout(IN:=NOT b2ThetaDriveReady OR NOT bSSLDriveReady,PT:=tEnableMotorTimeoutTime);

            // Are both drives reporting that they are ready?
            IF b2ThetaDriveReady AND bSSLDriveReady THEN
                iEnableMotorState := iEnableMotorState + 1;
                tonEnableMotorTimeout(IN:=FALSE);
            ELSIF tonEnableMotorTimeout.Q THEN
                IF NOT Main.M2.bError OR Main.M1.bError THEN
                    Main.M2.bError := TRUE;
                    Main.M1.bError := TRUE;
                    IF NOT b2ThetaDriveReady THEN
                        Main.M2.sCustomErrorMessage := 'Move failed because motor drive did not get ready status before timeout.';
                        Main.M1.sCustomErrorMessage := 'Move failed because 2 theta motor drive did not get ready status before timeout.';
                    ELSE
                        Main.M1.sCustomErrorMessage := 'Move failed because motor drive did not get ready status before timeout.';
                        Main.M2.sCustomErrorMessage := 'Move failed because SSL motor drive did not get ready status before timeout.';
                    END_IF
                END_IF
                iEnableMotorState := 0;
            END_IF
        3: // Allow the move execution to begin
            rtExecuteMove(CLK:=TRUE);
            IF rtExecuteMove.Q THEN
                Main.M2.bExecute := TRUE;
            END_IF
            tonEnableMotorTimeout(IN:=NOT Main.M2.bBusy,PT:=T#100ms);
            IF tonEnableMotorTimeout.Q THEN
                iEnableMotorState := iEnableMotorState + 1;
            END_IF
    ELSE
        iEnableMotorState := 0;
    END_CASE
ELSE
    Main.M2.bEnable := TRUE;
    Main.M1.bEnable := TRUE;
END_IF

fb2ThetaStepper(stMotionStage:=Main.M2);
END_ACTION

END_PROGRAM

// ---- POUs/PRG_SSL.TcPOU

PROGRAM PRG_SSL
VAR
    fb_SSL_Motor : FB_MotionStage;
    (*EPS Limit switches*)
    {attribute 'TcLinkTo' := 'TIIB[EL1004_02_03]^Channel 2^Input'}
    bLimitBackwardEnable AT %I* :BOOL;
    {attribute 'TcLinkTo' := 'TIIB[EL1004_02_03]^Channel 3^Input'}
    bLimitForwardEnable AT %I* :BOOL;
    {attribute 'pytmc' := 'pv: QRIX:SPCA:COUPLED'}

    bExecuteCouple: BOOL := FALSE;
    bExecuteDecouple: BOOL := FALSE;

    bInit : BOOl := TRUE;

    // Function block to couple sliding seal motor motion to 2Theta motion
    fbSSLTo2ThetaCoupling: FB_GantryAutoCoupling;

    {attribute 'TcLinkTo' := '	.Count := TIID^Device 2 (EtherCAT)^Rack#1A-01 Coupler (EK1100)^Rack#1A-06 ENC_2Th (EL5042)^FB Inputs Channel 1^Position'}
    stRenishawAbsEncMaster: ST_RenishawAbsEnc;

    {attribute 'TcLinkTo' := 'TIID^Device 2 (EtherCAT)^B950-233-WALL-S-R01-DRL-01^EL5042_02_02^FB Inputs Channel 1^Position'}
    nRenishawAbsEncSlaveCounts AT %I*: ULINT; // Connect to encoder "Position" inputULINT
    fSlaveCountsToMasterCountsScalingFactor: LREAL;
    fRenishawAbsEncSlaveCountsInMasterScale: LREAL;
    nRenishawAbsEncSlaveCountsInMasterScale: ULINT;
    stRenishawAbsEncSlave: ST_RenishawAbsEnc;

    nGantryTolerance: LINT;
    fAngleOffset: LREAL;


    {attribute 'pytmc' := '
        pv: QRIX:SSL2ThetaDegTol
        io: io
    '}
    fAngleTolerance: REAL := 0.2;

    {attribute 'pytmc' := '
        pv: QRIX:SSL2ThetaPosDiff
        io: i
    '}
    fPosDiff: REAL;

    fbExtSetPointGenEnable: MC_ExtSetPointGenEnable;
    fbExtSetPointGenDisable: MC_ExtSetPointGenDisable;

    {attribute 'pytmc' := '
        pv: QRIX:bRealignCouple
        io: io
    '}
    bRealignCouple: BOOL;
    {attribute 'pytmc' := '
        pv: QRIX:iRealignStep
        io: i
    '}
    iRealignStep: UINT := 0;
    {attribute 'pytmc' := '
        pv: QRIX:bRealignSpeed
        io: io
    '}
    fRealignSpeed: LREAL := 0.05;
    rtStopSSL: R_TRIG;
    tonRealignCoupleTimeout: TON;
    timeRealignTimeout: TIME;
    bFullyDecouple: BOOL;

    EL7047_02_01_SSL_Status AT %I*: USINT;
    EL7047_02_01_SSL_Status_to_NC AT %Q*: USINT;

END_VAR


IF bInit THEN
    bInit := FALSE;
    Main.M1.bPowerSelf := TRUE;
    Main.M1.bHardwareEnable := TRUE;
    Main.M1.nBrakeMode := ENUM_StageBrakeMode.NO_BRAKE;
    Main.M1.nEnableMode := ENUM_StageEnableMode.NEVER;
END_IF

// Due to bug in SSL drive, ready bit is not being reported properly. This will tie the ready bit to the floating status.
EL7047_02_01_SSL_Status.1 := GVL_Sensor.bFloating;
EL7047_02_01_SSL_Status_to_NC := EL7047_02_01_SSL_Status;

// Set the encoder counts at the zero position
// CHOOSING TO SET THE COUNTS IN UNITS OF THE SCALE OF THE PRIMARY AXIS ENCODER.
// THE VIRTUAL LIMIT SWITCH FUNCTION BLOCK IN THE GANTRY AUTOCOUPLING FB ASSUMES
// THAT THE ENCODERS HAVE THE SAME SCALE. HOWEVER IN THIS CASE, THEY DO NOT HAVE
// THE SAME SCALE. IN ORDER TO COMPARE THEM USING THE GANTRY FB, THE SECONDARY
// AXIS ENCODER COUNTS HAVE TO BE SCALED TO MATCH THE PRIMARY AXIS ENCODER COUNTS.
fSlaveCountsToMasterCountsScalingFactor := Main.M1.stAxisParameters.fEncScaleFactorInternal / Main.M2.stAxisParameters.fEncScaleFactorInternal;
fRenishawAbsEncSlaveCountsInMasterScale := ULINT_TO_LREAL(nRenishawAbsEncSlaveCounts) * fSlaveCountsToMasterCountsScalingFactor;
nRenishawAbsEncSlaveCountsInMasterScale := LREAL_TO_ULINT(fRenishawAbsEncSlaveCountsInMasterScale);
stRenishawAbsEncSlave.Count := nRenishawAbsEncSlaveCountsInMasterScale;

// Going to use 90 degree position as the reference position because the Ref value is an unsigned value. This makes it so I
// can't set the reference to actual 0 because that requires a negative number.
stRenishawAbsEncMaster.Ref := LREAL_TO_ULINT((90.0 - Main.M2.stAxisParameters.fEncOffset) / Main.M2.stAxisParameters.fEncScaleFactorInternal);
stRenishawAbsEncSlave.Ref := LREAL_TO_ULINT((90.0 - Main.M1.stAxisParameters.fEncOffset) / Main.M1.stAxisParameters.fEncScaleFactorInternal * fSlaveCountsToMasterCountsScalingFactor);

// Compute the gantry tolerance
// Tolerance = X degrees
// 0.000003001664895 deg/count => For 0.1 deg tolerance then 0.1 deg / 0.000003001664895 deg/count = 33315 counts for 0.1 deg
nGantryTolerance := LREAL_TO_LINT(fAngleTolerance / Main.M2.stAxisParameters.fEncScaleFactorInternal);

fAngleOffset := LINT_TO_LREAL(
        ( ULINT_TO_LINT(stRenishawAbsEncMaster.Count) - ULINT_TO_LINT(stRenishawAbsEncMaster.Ref) ) -
        ( ULINT_TO_LINT(stRenishawAbsEncSlave.Count) - ULINT_TO_LINT(stRenishawAbsEncSlave.Ref) )
    ) * Main.M2.stAxisParameters.fEncScaleFactorInternal;

// AutoCoupling
fbSSLTo2ThetaCoupling(	nGantryTol 			:= nGantryTolerance,
                        Master				:= Main.M2,
                        MasterEnc			:= stRenishawAbsEncMaster,
                        Slave				:= Main.M1,
                        SlaveEnc			:= stRenishawAbsEncSlave,
                        bExecuteCouple 		:= bExecuteCouple,
                        bExecuteDecouple 	:= bExecuteDecouple,
);

// Calculate twice the expected amount of time to make the realignment move.
timeRealignTimeout := LREAL_TO_TIME(abs(Main.M1.stAxisStatus.fActPosition - Main.M2.stAxisStatus.fActPosition) / fRealignSpeed * 3.0 * 1000.0);
tonRealignCoupleTimeout(IN:=bRealignCouple,PT:=timeRealignTimeout);
CASE iRealignStep OF
    0:
        IF bRealignCouple THEN
            iRealignStep := 1;
        END_IF
    1:
        // Step 1: If the gantry is already coupled, the motor is not busy, and it is enabled, then decouple the axes.
        IF fbSSLTo2ThetaCoupling.bGantryAlreadyCoupled AND NOT Main.M1.bBusy AND NOT Main.M1.bError THEN
            bExecuteDecouple := TRUE;
            iRealignStep := 2;
        ELSIF NOT fbSSLTo2ThetaCoupling.bGantryAlreadyCoupled AND NOT Main.M1.bBusy AND NOT Main.M1.bError THEN
            iRealignStep := 2;
        END_IF
    2:
        // Step 2: If the gantry is no longer coupled, the motor is not busy, and it is enabled, then reset the decouple command and
        //         command the axis to align the SSL motor to the 2Theta motor. Set the bTriedToRealign bit to true to record that
        //         the realign sequence is what commanded the move.
        IF NOT fbSSLTo2ThetaCoupling.bGantryAlreadyCoupled AND NOT Main.M1.bBusy AND NOT Main.M1.bError THEN
            bExecuteDecouple := FALSE;
            Main.M1.fPosition := Main.M2.stAxisStatus.fActPosition;
            Main.M1.fVelocity := fRealignSpeed;
            Main.M1.bMoveCmd := TRUE;
            iRealignStep := 3;
        END_IF
    3:
        // Step 3: Wait for the SSL motor to reach the busy status, then proceed.
        IF Main.M1.bBusy THEN
            iRealignStep := 4;
        END_IF
    4:
        // Step 4: If the SSL motor is no longer busy (finished or errored or stopped) then recouple the SSL motor to
        //         the 2Theta motor.
        IF NOT Main.M1.bBusy AND NOT Main.M1.bError THEN
            bExecuteCouple := TRUE;
            iRealignStep := 5;
        END_IF
    5:
        // Step 5: If the motors are coupled again then reinitialize the bits to
        //         get them ready for another realignment attempt in the future.
        IF fbSSLTo2ThetaCoupling.bGantryAlreadyCoupled THEN
            iRealignStep := 0;
            bRealignCouple := FALSE;
            bExecuteDecouple := FALSE;
            bExecuteCouple := FALSE;
            tonRealignCoupleTimeout(IN:=FALSE);
        ELSE
            iRealignStep := 4;
        END_IF
END_CASE

// Timeout: In case something bad happens, have the timeout timer in place to reset the bits to guarantee we do not get
//          stuck in this recoupling and alignment sequence.
// If coupled axis fails to move due to axis not ready, may need to force the SSL motor ready status to TRUE. Then is allows it to move.
// seems like some sort of bug with decoupling/coupling the axes too much.
IF bRealignCouple AND tonRealignCoupleTimeout.Q THEN
    IF fbSSLTo2ThetaCoupling.bGantryAlreadyCoupled OR Main.M1.bError THEN
        iRealignStep := 0;
        bRealignCouple := FALSE;
        bExecuteDecouple := FALSE;
        bExecuteCouple := FALSE;
        tonRealignCoupleTimeout(IN:=FALSE);
    ELSIF NOT Main.M1.bBusy THEN
        bExecuteCouple := TRUE;
    END_IF
END_IF

fPosDiff := Main.M1.stAxisStatus.fActPosition - Main.M2.stAxisStatus.fActPosition;

fb_SSL_Motor(stMotionStage:=Main.M1);

END_PROGRAM

// ---- Spectometer Arm POUs/PRG_DET_ARM.TcPOU

PROGRAM PRG_DET_ARM
VAR
    bInit: BOOL := TRUE;
    bExecuteCouple: BOOL := FALSE;
    bExecuteDecouple: BOOL := FALSE;

    fbMotionYF1: FB_MotionStage;
    fbMotionYF2: FB_MotionStage;
    fbMotionZF: FB_MotionStage;
    fbAutoCoupling: FB_GantryAutoCoupling;

    {attribute 'TcLinkTo' := '	.Count := TIIB[BOX-06 ENC_ZDC_YF1 (EL5042)]^FB Inputs Channel 2^Position'}
    stRenishawAbsEncMaster: ST_RenishawAbsEnc;
    {attribute 'TcLinkTo' := '	.Count := TIIB[BOX-07 ENC_YF2_ZF (EL5042)]^FB Inputs Channel 1^Position'}
    stRenishawAbsEncSlave: ST_RenishawAbsEnc;

    tonDelay: TON;
    tonDelay2: TON;
    rtDelay: R_TRIG;
    bRunTimer: BOOL;
    nState: INT := -1;
    bDisableStateMachine: BOOL;


    {attribute 'TcLinkTo' := '.nMicrostepCounter := TIID^Device 2 (EtherCAT)^BOX-01 Coupler (EK1100)^BOX-20 DR_YF1 (EL7047)^ENC Status compact^Counter value;
                              .bCounterOverflow  := TIID^Device 2 (EtherCAT)^BOX-01 Coupler (EK1100)^BOX-20 DR_YF1 (EL7047)^ENC Status compact^Status^Counter overflow;
                              .bCounterUnderflow := TIID^Device 2 (EtherCAT)^BOX-01 Coupler (EK1100)^BOX-20 DR_YF1 (EL7047)^ENC Status compact^Status^Counter underflow'}
    fbMeasureReferenceVelocity: FB_MeasureReferenceVelocity;
END_VAR


IF bInit THEN
    bInit := FALSE;
    bExecuteCouple := TRUE;

    Main.M25.nBrakeMode := ENUM_StageBrakeMode.NO_BRAKE;
    Main.M25.bHardwareEnable := TRUE;
    Main.M25.bPowerSelf := TRUE;
    Main.M25.fVelocity := 0.1;

    Main.M26.nBrakeMode := ENUM_StageBrakeMode.NO_BRAKE;
    Main.M26.bHardwareEnable := TRUE;
    Main.M26.bPowerSelf := TRUE;
    Main.M26.fVelocity := 0.1;

    Main.M27.nBrakeMode := ENUM_StageBrakeMode.IF_ENABLED;
    Main.M27.bHardwareEnable := TRUE;
    Main.M27.bPowerSelf := TRUE;
    Main.M27.fVelocity := 0.1;

